(* CODESYS project unilib.library
   Company: Beckhoff Automation GmbH & Co. KG
   DefaultNamespace: TC3_UniLib
   Version: 1.2.10.2
   Placeholder: UniLib Gruppe 11
   Author: Christian Frickenstein, Bernhard Edenfeld, Benedikt Daut
   Description: Zentrale Bausteine für die Programmierung in der Gruppe 11. Hinweise zu den Versionsnummern: 1. Zahl: Grundsätzliche Version für TwinCAT3, 2. Zahl: für die verschiedenen Varianten. Nicht abwärtskompatibel, 3. Zahl: Neue Bausteine oder Funktionen hinzugefügt, aber abwärtskompatibel ggf. neue Eingänge oder Umbenennungen. 4. Zahl: Bugfixes, bedingungslos abwärtskompatibel
   Title: UniLib Gruppe 11

Project tree, tasks and I/O mapping:
  libraries: Tc2_EtherCAT, * (Beckhoff Automation GmbH); Tc2_IoFunctions, * (Beckhoff Automation GmbH); Tc2_MC2, * (Beckhoff Automation GmbH); Tc2_MC2_Drive, * (Beckhoff Automation GmbH); Tc2_SerialCom, * (Beckhoff Automation GmbH); Tc2_Standard, * (Beckhoff Automation GmbH); Tc2_System, * (Beckhoff Automation GmbH); Tc2_Utilities, * (Beckhoff Automation GmbH); Tc3_JsonXml, * (Beckhoff Automation GmbH); Tc3_Module, * (Beckhoff Automation GmbH)
  DUTs/
    ComPort/
      data type E_ComPortHardware
      data type E_ComPortKlemmenBytes
      data type E_ComPortProtokoll
      data type ST_ComPortFlags
      data type ST_ComPortInData
      data type ST_ComPortIntBuffer
      data type ST_ComPortOptions
      data type ST_ComPortOptionsIntern
      data type ST_ComPortOutData
      data type ST_ComPortStringBuffer
      data type ST_InInfoDataSerielleKlemme
      data type ST_MethodResult
    DiagEL2904/
      data type ST_EL2904Diag
      data type ST_EL2904Temp
    EAP/
      data type ST_EAP_Kommunikation
      data type ST_EAP_Receive
      data type ST_EAP_Send
      data type ST_StepCtrl
      data type ST_StepPara
      data type ST_TEMP_EAP_TEST
      data type ST_TempEAPDaten
      data type ST_TwinSAFE_Connection
      data type U_EAP_Kommunikation
    HMI_DataExchange/
      data type ST_HMIDataExchange
    HMI_Grundstrukturen/
      data type ST_HandFktHMI
      data type ST_OP_HMI
      data type ST_OP_Visual
    HMI_Meldungen/
      Meldelisten/
        Allgemein/
          data type ST_MeldTextAllgm
        InternAchsen/
          data type ST_MeldAchsfehler
          data type ST_MeldAchsGruppe
        InternEinspeis/
          data type ST_MeldAuffrischKlemme
          data type ST_MeldEinspeisKlemme
        InternSafety/
          data type ST_MeldKlemme
          data type ST_MeldSafetyFBErrors
          data type ST_MeldSafetygruppe
          data type ST_MeldSafetyOuts
        InternSchaltschrank/
          data type ST_MeldElektrSichg
          data type ST_MeldKlimaGeraet
          data type ST_MeldMotSchutzS
          data type ST_MeldSchaltNetzT
          data type ST_MeldSichgAutom
          data type ST_MeldThermoUeberw
          data type ST_MeldUSV
        InternSchutzbereich/
          data type ST_MeldNotHalt
          data type ST_MeldSchutzbereichOffen
          data type ST_MeldSichLichtg
          data type ST_MeldStHLuft
          data type ST_MeldTuerFrgBremsentest
          data type ST_MeldWartgTuer
        InternSonstiges/
          data type ST_MeldADS_ExchangeError
          data type ST_MeldADSKommError
          data type ST_MeldBetriebsdruck
          data type ST_MeldDatenanf
          data type ST_MeldEAPKommError
          data type ST_MeldEtherCAT
          data type ST_MeldGrundstellung
          data type ST_MeldIOLinkKlemme
        UniAnstg/
          data type ST_MeldAchsKontrl
          data type ST_MeldTextUniAchs
          data type ST_MeldTextUniAktr
          data type ST_MeldTextUniAntr
          data type ST_MeldTextUniWkzg
          data type ST_MeldTextUniZyli
        data type ST_MeldAchsList
        data type ST_MeldEAPList
        data type ST_MeldIOLinkList
        data type ST_MeldKommunikationsList
        data type ST_MeldPotentialList
        data type ST_MeldSafetyList
        data type ST_MeldSchaltSchrList
        data type ST_MeldSchutzberList
        data type ST_MeldSeriellComPort
      data type ST_0100_Meldungen
      data type ST_ParamHMIMaschine_Beispiel
    HMI_Parameter/
      data type ST_UniAchsAnstgParam
      data type ST_UniAntrAnstgParamAggr
      data type ST_UniAntrAnstgParamAggrHF
      data type ST_UniAntrAnstgParamTrsp
    HMI_UniAnstgHandFktMeldungen/
      data type E_AnstgArtUniAktr
      data type E_AnstgArtUniAntr
      data type E_AnstgArtUniWkzg
      data type E_AnstgArtUniZyli
      data type E_AntriebTyp
      data type E_ZylinderTyp
      data type ST_UniAchsAnstg
      data type ST_UniAktrAnstg
      data type ST_UniAntrAnstg
      data type ST_UniBaustein
      data type ST_UniGrdstlgAbl
      data type ST_UniWkzgAnstg
      data type ST_UniZyliAnstg
    Meldebox/
      data type ST_MessageBox
    NcAchsen/
      data type ST_AchsAuftrg
      data type ST_AchsFreigb
      data type ST_AchsGrdfkt
      data type ST_AchsInOut
      data type ST_AchsKoppln
      data type ST_AchsMeldg
      data type ST_AchsParam
      data type ST_AchsStatus
      data type ST_NcAchsen
    SEW/
      data type ST_SEWInput
      data type ST_SEWOutput
    TwinSAFE/
      data type E_SafetyType
      data type ST_TwinSAFE_Conn_Info
      data type ST_TwinSAFE_ConnInfoBasis
      data type ST_TwinSAFE_FB_Info
      data type ST_TwinSAFE_Group_Info
      data type ST_TwinSAFEConnInfo4Byte
      data type ST_TwinSAFEConnInfo5Byte
      data type ST_TwinSAFEKlemmenInfo
    data type ST_TimeStamp
    data type ST_TimeStruct
  GVLs/
    global variables AllgemeineParameter
    global variables ComPortParameterliste
    global variables GlobalVar_Allgemein
    global variables GlobalVar_Farben
    global variables GlobalVar_TestMeld
  POUs/
    ComPort_2_0_1_0/
      function F_ComReceiveBarcode [ST]
      function F_ComSendBarcode [ST]
      function block FB_ComBackground [ST]
      function block FB_ComConfig [ST]
      function block FB_ComMain [ST]
      function block FB_ComPortOld [ST]
    ComPort_3_0_1_0/
      function block FB_ComPort [ST]: ccl_Backround, ccl_Main, ccl_Messages, ccl_Receive, FB_init, nccl_Config, nccl_PrepareSendBarcode, nccl_ReceiveBarcode, nccl_Reset, nccl_Send, P_bDatenVorhanden, P_stEmpfangeneDaten, P_stEmpfangenerString
      data type ST_MeldComPort
    DiagSafety/
      function block FB_DiagEL2904 [ST]: act_Diag, act_DiagObjekte
      function block FB_DiagEL2912 [ST]: act_Diag
      function block FB_TwinSAFE_Conn_Info [ST]: act_Diag, act_State, actInfo
      function block FB_TwinSAFE_FBs_Info [ST]: act_Diag, act_State, actInfoAND, actInfoConnectionShutDown, actInfoDecoupler, actInfoEDM, actInfoEStop, actInfoMON, actInfoMuting, actInfoOPMode, actInfoOR, actInfoRS, actInfoSR, actInfoTOF, actInfoTON, actInfoTwoHand
      function block FB_TwinSAFE_Group_Info [ST]: act_State, actInfo
      function block FB_TwinSAFEConnInfo [ST]: act_Diag, act_State, actInfo
      function block FB_TwinSAFEConnInfo4Byte [ST]: a_Info, b_State, c_Diag
      function block FB_TwinSAFEConnInfo4Byte_1 [ST]: a_Info, b_State, c_Diag
      function block FB_TwinSAFEConnInfo5Byte [ST]: a_Info, b_State, c_Diag
      function block FB_TwinSAFEConnInfo5Byte_1 [ST]: a_Info, b_State, c_Diag
      function block FB_TwinSAFEConnInfoBasis [ST]: a_Info, b_State, c_Diag
      function block FB_TwinSAFEFBsInfo [ST]: act_Diag, act_State, actInfoAND, actInfoConnectionShutDown, actInfoDecoupler, actInfoEDM, actInfoEStop, actInfoMON, actInfoMuting, actInfoOPMode, actInfoOR, actInfoRS, actInfoSR, actInfoTOF, actInfoTON, actInfoTwoHand
      function block FB_TwinSAFEGroupInfo [ST]: act_State, actInfo
      function block FB_TwinSAFEKlemmeInfo [ST]: a_Initialisierung, b_Ablauf, c_EL6900, c_EL6910, d_EK1914, d_EL1904, d_EL1918, d_EP1908, d_EP1918, d_EP1957, e_EL2904, e_EL2911, e_EL2912, e_EP2918, f_AX5805, f_AX5806
    Diverse/
      function F_Skalierung [ST]
      function F_Switchbyte [ST]
      function block FB_Blinker [ST]
      function block FB_ElectronicFuseIOLink [ST]: a_GetCurrent, b_GetStatus, z_Message, z_Output
      function block FB_SafetyElementAnz [ST]
      function block FB_UsvStatus [ST]
      function block FB_WartgTuer [ST]: a_TuerEntrieg, b_AutomHalt
      function block FB_WartgTuerMeld [ST]: a_TuerEntrieg, b_AutomHalt, z_Meld
      function block FB_WartgTuerMeldAnz [ST]: a_TuerEntrieg, b_AutomHalt, c_Anzeige, z_Meld
    EAP/
      function block FB_EAP_Kommunikation [ST]: _00_Init, _02_TwinSAFE, m_DatenBereitstellen, m_Receive, m_Send, m_Senden
      function block FB_EAP_Kommunikation_V2 [ST]: _02_TwinSAFE, _07_Senden_Empfangen, _10_Meldungen, m_Senden
      function block FB_StepUebw [ST]
    EtherCATDiagnose/
      data type E_EcCommState
      function block FB_EtherCATDiag [ST]: a_GetSlaveAdresses, b_GetSlaveStates, c_GetTopoDataLen, d_GetTopoData, e_ScanSlaves, f_GetSlaveIdentity, g_GetSlaveName, h_GetScannedSlaveName, i_ErrorMessage, j_CheckMasterDevState, k_SlaveErrorMessage
      function block FB_EtherCATFrameDiag [ST]
      function block FB_IoLinkFehler [ST]
      data type ST_EcMasterDevState
      data type ST_EcPortAddr
      data type ST_SlaveState
      data type ST_SlaveStateInfo
      data type ST_SlaveStateInfoScanned
      data type ST_TopologyData
    Grundstellung/
      function block FB_UniGrdstlgAbl [ST]: a_AnAbwahl, b_StepAblauf, y_ZustAnzg, z_HinwMeld
      function block FB_UniGrdstlgAblBereich [ST]: a_AnAbwahl, b_StepAblauf, y_ZustAnzg, z_HinwMeld
      function block FB_UniGrdstlgAblGesamt [ST]: a_AnAbwahl, b_StepAblauf, y_ZustAnzg, z_HinwMeld
    Logging/
      function F_AdsErrorIdToString [ST]
      function F_TimeStruct [ST]
      function block FB_LogToFile [ST]
      function block FB_StepHistory [ST]
      function block FB_TaktzeitAuswert [ST]: a_DateiSchreiben
    MeldTest/
      function block FB_MeldTestAllgemein [ST]
    Time/
      function block FB_Zeitstempel [ST]
    UniBausteine/
      function block FB_LaufzMeldg [ST]
      function block FB_LaufzMeldgAktr [ST]
      function block FB_UniAchsAnstg [ST]: a_Standard, w_InOutNc, y_ZustAnzg, z_FehlMeld
      function block FB_UniAktrAnstg [ST]: a_Standard, x_AusgZuw, y_ZustAnzg, z_FehlMeld
      function block FB_UniAntrAnstg [ST]: a_Aggregat, b_Transport, c_Verstellg, x_AusgZuw, y_ZustAnzg, z_FehlMeld
      function block FB_UniAntrAnstgSEW [ST]: a_Aggregat, b_Transport, c_Verstellg, d_EilSchleich, u_AggEinlZykl, v_AggBetrZykl, w_InOutSEW, x_AusgZuw, y_ZustAnzg, z_FehlerAusw, z_FehlMeld
      function block FB_UniAntrAnstgSEW_IO [ST]: a_Aggregat, b_Transport, c_Verstellg, d_EilSchleich, u_AggEinlZykl, v_AggBetrZykl, w_InOutSEW, x_AusgZuw, y_ZustAnzg, z_FehlMeld
      function block FB_UniHydrAnstgHubb [ST]: a_Standard, x_AusgZuw, y_ZustAnzg, z_FehlMeld
      function block FB_UniWkzgAnstg [ST]: a_Standard, b_PulsUebw, x_AusgZuw, y_ZustAnzg, z_FehlMeld
      function block FB_UniZyliAnstg [ST]: a_Standard, b_MittelStellung, c_TestMode, x_AusgaengeZuweisen, y_ZustaendeAnzeigen, z_FehlerMeldung
*)

// DUTs/ComPort/E_ComPortHardware
{attribute 'qualified_only'}
// Comportdefinition der Hardware
TYPE E_ComPortHardware:(
	cComportPc,	// Der Comport kommt aus einem PC
	cComportKL,	// Der Comport kommt von einer KL-Klemme
	cComportEL	// Der Comport kommt von einer EL-Klemme
);
END_TYPE

// DUTs/ComPort/E_ComPortKlemmenBytes
{attribute 'qualified_only'}
// Größe des Byte-Streams aus der Hardware-Verbindung
TYPE E_ComPortKlemmenBytes:(
	cComport3Bytes,	// Der Komport liefert einen Byte-Stream von 3 Byte, alte Klemmen
	cComport5Bytes,	// Der Komport liefert einen Byte-Stream von 5 Byte, alte Klemmen
	cComport22Bytes	// Der Komport liefert einen Byte-Stream von 22 Byte, aktueller Standard
);
END_TYPE

// DUTs/ComPort/E_ComPortProtokoll
{attribute 'qualified_only'}
// Protokoll, wie der empfangene Byte-Stream ausgewertet werden soll
TYPE E_ComPortProtokoll :(
	cProtokollNone,	// Protokoll, wie der Byte-Stream ausgewertet werden soll. Hier wird der Byte-Stream dirket ausgegeben
	cProtokollData,	// Protokoll, wie der Byte-Stream ausgewertet werden soll. Hier wird der Byte-Stream dirket ausgegeben
	cProtokollDirect,	// Protokoll, wie der Byte-Stream ausgewertet werden soll. Hier wird der Byte-Stream dirket ausgegeben
	cProtokollBarcode,	// Protokoll, wie der Byte-Stream ausgewertet werden soll. Hier wird der Byte-Stream als STRING ausgegeben
	cProtokollP3964	// Protokoll, wie der Byte-Stream ausgewertet werden soll. Hier wird der Byte-Stream im P3964-Format ausgegeben
);
END_TYPE

// DUTs/ComPort/ST_ComPortFlags
TYPE ST_ComPortFlags :
STRUCT
	(* Konfiguration *)
	bConfigFlag		: BOOL;			(* Anstossen der Schnittstellenkonfiguration *)

	(* Schnittstellenpuffer loeschen *)
	bResetFlag		: BOOL;			(* Loeschen des internen Schnittstellenpuffers *)

	(* Empfangen *)
	bRxFlag			: BOOL;			(* Anstossen der Datenauswertung bei Empfang *)
	bWaitQuitFlag	: BOOL;			(* Quittieren der neg. Flanke von VB*)

	(* Senden *)
	bTxFlag			: BOOL;			(* Anstossen des Sendens *)
END_STRUCT
END_TYPE

// DUTs/ComPort/ST_ComPortInData
// Datentyp für die Verbindung zur Hardwareschnittstelle. Für alle Byte-Streamtypen. Nur eine Verbindung nutzen!!!
TYPE ST_ComPortInData :
STRUCT
	stKlemmeIn3B	: Tc2_SerialCom.KL6inData;	// Inputdaten für 3Byte-Klemmen
	stKlemmeIn5B	: Tc2_SerialCom.KL6inData5B;	// Inputdaten für 5Byte-Klemmen
	stKlemmeIn22B	: Tc2_SerialCom.KL6inData22B;	// Inputdaten für 22Byte-Klemmen
	stPCIn			: Tc2_SerialCom.PcComInData;	// Inputdaten für PC-Verbindung
	stInfoData		: ST_InInfoDataSerielleKlemme;	// Infodaten, sollten mit einer Klemme verküpft werden um sie automatisch zu parametrieren
END_STRUCT
END_TYPE

// DUTs/ComPort/ST_ComPortIntBuffer
// Datentyp für den Internen Byte-Stream
TYPE ST_ComPortIntBuffer :
STRUCT
	arrData	: ARRAY [0..cBufferSize_IntBuffer] OF UINT;	// Interner Puffer für die Empfangenen Bytes
END_STRUCT
END_TYPE

// DUTs/ComPort/ST_ComPortOptions
// Optionen für den Comport
TYPE ST_ComPortOptions:
STRUCT
	nId				: UINT;	// Allgemeine Nummerierung
	
	nBaudrate  		: UINT;	// 1200, 2400, 4800, 9600, 19200
	nDatenbits		: UINT;	// 7, 8
	nStopbits 		: UINT;	// 1, 2
	nParitaet 		: INT;	// 0: keine Parität, 1: gerade(even) Parität, 2: ungerade(odd) Parität
	nHandshake		: INT;	// 0: Kein Handshake, 1: RTS/CTS, 2: XON/XOFF
	
	eProtokoll 		: E_ComPortProtokoll;	// 0: kein, 1: Daten, 2: Direkt, 3: Barcode, 4: 3964
	nPrefix 			: UINT;	// 0: kein, 2: STX
	nSuffix1 		: UINT;	// 0: kein, 13: CR, 3: ETX, 4: EOT 
	nSuffix2 		: UINT;	// 0: kein, 10: LF
	nTimeout 		: UINT;	// Maximale Zeit zwischen zwei Zeichen, bei String oder Barcodeempfang
	nLength			: INT;	// Anzahl der zu empfangenen Zeichen, incl. Präfix und Suffix
	
	ePort				: E_ComPortHardware;	// 0: PC, 1: Klemme, 2: E-Klemme
	eComPortBytes	: E_ComPortKlemmenBytes;	// 0: 3 Bytes, 1: 5 Bytes, 2: 22 Bytes
	nAktiv			: UINT;	// 0: Schnittstelle nicht aktiv, 1: Schnittstelle aktiv
	nCommVB			: UINT;	// 0: DotNet als Applikation, 1: VisualBasic als Applikation
END_STRUCT
END_TYPE

// DUTs/ComPort/ST_ComPortOptionsIntern
// Datentyp für die Internen Optionen
TYPE ST_ComPortOptionsIntern :
STRUCT
	nPrefix			: BYTE;	// Präfix als ASCII-Zeichen
	sPrefix			: STRING(10);	// Präfix als String
	nLenPrefix		: BYTE;	// Länge des Prefixes

	arrSuffix		: ARRAY[1..2] OF BYTE;	// Suffix als ASCII-Array
	sSuffix			: STRING(10);	// Suffix als String
	nLenSuffix		: BYTE;	// Länge des Suffixes

	tTimeTimeout	: TIME;	// Maximale Zeit zwischen zwei Zeichen, bei String oder Barcodeempfang
   nLength			: INT;	// Anzahl der zu empfangenen Zeichen, incl. Präfix und Suffix
END_STRUCT
END_TYPE

// DUTs/ComPort/ST_ComPortOutData
// Datentyp für die Verbindung zur Hardwareschnittstelle. Für alle Byte-Streamtypen. Nur eine Verbindung nutzen!!!
TYPE ST_ComPortOutData :
STRUCT
	stKlemmeOut3B	: KL6outData;	// Outputdaten für 3Byte-Klemmen (obsolet)
	stKlemmeOut5B	: KL6outData5B;	// Outputdaten für 5Byte-Klemmen	(obsolet)
	stKlemmeOut22B	: KL6outData22B;	// Outputdaten für 22Byte-Klemmen (standard)
	stPCOut			: PcComOutData;	// Outputdaten für PC-Verbindungen
END_STRUCT
END_TYPE

// DUTs/ComPort/ST_ComPortStringBuffer
// Datentyp: Empfangener Stream als STRING in variabler Größe
TYPE ST_ComPortStringBuffer :
STRUCT
	sData	: STRING(cBufferSize_StringBuffer);	// variable STRING-Variable
END_STRUCT
END_TYPE

// DUTs/ComPort/ST_InInfoDataSerielleKlemme
// Datentyo zur ADS-Verbindung mit der Klemme
TYPE ST_InInfoDataSerielleKlemme :
STRUCT
	stADSNetId	: Tc2_System.T_AmsNetIdArr;	// ADS-NETID 172.50.12.1.1.1 oder ähnlich
	nADSPort		: UINT;	// ADS-Port: 1002 oder höher
END_STRUCT
END_TYPE

// DUTs/ComPort/ST_MethodResult
// Ergebnisvariable einer Methode
TYPE ST_MethodResult :
STRUCT
	bBusy		: BOOL;	// Methode ist aktiv und noch nicht abgearbeitet
	bDone		: BOOL;	// Methode ist abgearbeitet
	bError	: BOOL;	// Error bei Bearbeitung aufgetreten 
	nErrorId	: INT;	//	Error als ID
	sError	: STRING;	// Error als Klartext
END_STRUCT
END_TYPE

// DUTs/DiagEL2904/ST_EL2904Diag
// OBSOLET, wenn man FB_TwinSAFEKlemmenInfo benutzt
TYPE ST_EL2904Diag :
STRUCT
	nDummyData1								:ARRAY[0..10] OF UINT;

(* Error at the outputs *)
	nErrorOutputs							:UINT;

(* Supply error *)
	nSupplyError							:UINT;

(* Temperature error *)
	nTemperatureError						:UINT;

	nDummyData2								:ARRAY[0..1] OF UINT;

END_STRUCT
END_TYPE

// DUTs/DiagEL2904/ST_EL2904Temp
// OBSOLET, wenn man FB_TwinSAFEKlemmenInfo benutzt
TYPE ST_EL2904Temp :
STRUCT	
	nInternalTemperature1					:INT;	(* Temperature 1 [°C] *)
	nInternalTemperature2					:INT;	(* Temperature 2 [°C] *)
	nInternalTemperatureOutputs			:INT;	(* Temperature 2 [°C] *)
END_STRUCT
END_TYPE

// DUTs/EAP/ST_EAP_Kommunikation
{attribute 'pack_mode' := '0'}
TYPE ST_EAP_Kommunikation :
STRUCT
	KommBits				: DWORD;
	TeilID				: STRING(19);
	TeilStatus			: DWORD;		
	ZusatzInfo1			: DWORD;		
	ZusatzInfo2			: DWORD;		
	ZusatzInfo3			: DWORD;		
	ZusatzInfo4			: DWORD;		
	ZusatzInfo5			: DWORD;		
	ZusatzInfo6			: DWORD;		
	ZusatzInfo7			: DWORD;		
	ZusatzInfo8			: DWORD;		
	ZusatzInfo9			: DWORD;		
	ZusatzInfo10		: DWORD;		
	
	//71BYTE

END_STRUCT
END_TYPE

// DUTs/EAP/ST_EAP_Receive
TYPE ST_EAP_Receive :
STRUCT
	VarState		AT %I* : UINT;
	Quality		AT %I* : UINT;
	CycleIndex	AT %I* : UINT;
	VarData		AT %I* : U_EAP_Kommunikation; 
END_STRUCT
END_TYPE

// DUTs/EAP/ST_EAP_Send
TYPE ST_EAP_Send :
STRUCT
	FrameState	AT %I* : UINT;
	FrameCtrl	AT %Q* : UINT;
	VarState		AT %I* : UINT;
	VarCtrl		AT %Q* : UINT;
	VarData		AT %Q* : U_EAP_Kommunikation; 
END_STRUCT
END_TYPE

// DUTs/EAP/ST_StepCtrl
// SK20190724:
// StepControl entählt folgende Funktionalitäten:
//	-> Delayabfrage und -Ausgabe
//	-> fbStepHistory mit optionaler Status Eintragung
//	-> Variablen für die Schrittkette
// !!! <VarName>.fbHistory(IQ_StepPara := <VarName>.IQ); notwendig
TYPE ST_StepCtrl :
STRUCT
	IQ				: ST_StepPara;
	fbHistory	: FB_StepUebw;
END_STRUCT
END_TYPE

// DUTs/EAP/ST_StepPara
TYPE ST_StepPara :
STRUCT
	
	nStep			: INT;
	sStatus		: T_MaxString;
	I_tDelay		: TIME;		// Delayvorgabe			Timer läuft ab, wenn Step = oldStep
	Q_bDelay		: BOOL;		// Delay abgelaufen
	I_bAblaufIN	: BOOL;		//								Timer läuft ab, wenn I_bAblaufIN = TRUE
	I_tAblauf	: TIME;		// Delayvorgabe
	Q_bAblauf	: BOOL;		// Delay abgelaufen
	I_bReset		: BOOL;
	I_bSaveLog	: BOOL;

END_STRUCT
END_TYPE

// DUTs/EAP/ST_TEMP_EAP_TEST
TYPE ST_TEMP_EAP_TEST :
STRUCT
	tonStartDif			: TON;
	tonDifEAP			: TON;
	tonDifKabel			: TON;
	
	bStartDifEAP		: BOOL;
	bStartDifKabel		: BOOL;
	
	ftStartDif			: F_TRIG;
	ftStartEAP			: F_TRIG;
	ftStartKabel		: F_TRIG;
	rtStopMessung		: R_TRIG;

	
	bEAPSchneller		: BOOL;
	bKabelSchneller	: BOOL;
	bGleich				: BOOL;
	bAlleUnngleich		: BOOL;
	tZeitDif				: TIME;
	
	nEAPkeinSignal		: INT;	
	
	
	

END_STRUCT
END_TYPE

// DUTs/EAP/ST_TempEAPDaten
TYPE ST_TempEAPDaten :
STRUCT
	sTeilenummer		: STRING(19);	// Teilenummer 
	wStatus				: DWORD;			// Der Status des Teils
	wZusatzinfo1		: DWORD;			//	Zusätzliche Infos 1
	wZusatzinfo2		: DWORD;			// Zusätzliche Infos 2
	wZusatzinfo3		: DWORD;			// Zusätzliche Infos 3
	wZusatzinfo4		: DWORD;			// Zusätzliche Infos 4
	wZusatzinfo5		: DWORD;			// Zusätzliche Infos 5
	wZusatzinfo6		: DWORD;			// Zusätzliche Infos 6
	wZusatzinfo7		: DWORD;			// Zusätzliche Infos 7
	wZusatzinfo8		: DWORD;			// Zusätzliche Infos 8
	wZusatzinfo9		: DWORD;			// Zusätzliche Infos 9
	wZusatzinfo10		: DWORD;			// Zusätzliche Infos 10
END_STRUCT
END_TYPE

// DUTs/EAP/ST_TwinSAFE_Connection
TYPE ST_TwinSAFE_Connection :
STRUCT
	 
	I_nID				: INT;
	I_sConnName		: STRING;
	I_nGroupID		: INT;
	Q_bIn0			: BOOL;
	Q_bIn1			: BOOL;
	Q_bIn2			: BOOL;
	Q_bIn3			: BOOL;
	Q_bIn4			: BOOL;
	Q_bIn5			: BOOL;
	Q_bIn6			: BOOL;
	Q_bIn7			: BOOL;
	Q_bOut0			: BOOL;
	Q_bOut1			: BOOL;
	Q_bOut2			: BOOL;
	Q_bOut3			: BOOL;
	Q_bOut4			: BOOL;
	Q_bOut5			: BOOL;
	Q_bOut6			: BOOL;
	Q_bOut7			: BOOL;
	Q_bErrDiag		: BOOL;
	Q_bErrState		: BOOL;
	Q_sDiag			: STRING(255);
	Q_sState			: STRING(255);

END_STRUCT
END_TYPE

// DUTs/EAP/U_EAP_Kommunikation
TYPE U_EAP_Kommunikation :
UNION
	Komm	: ARRAY[1..71] OF BYTE;
	Data	: ST_EAP_Kommunikation;
END_UNION
END_TYPE

// DUTs/HMI_DataExchange/ST_HMIDataExchange
{attribute 'pack_mode' := '1'}
// TODO: muss in die BAAvalonLib wandern

TYPE ST_HMIDataExchange :
STRUCT
	bNewData			: BOOL;		// Trigger Variable Plc setzt = TRUE => Oberfläche setzt zurück (FALSE)
	nStatus			: DINT;		// 1 Ok / > 1 Fehler
	sData				: STRING;	// Daten die von Plc kommen Barcode, Bohrbilder, PersonalNummern
	nTyp				: INT;		// Zur weitern Differenzierung der Daten (z.B. 1:Teilebarcode/2:Stapelbarcode)
	sSource			: STRING;	// Quelle von der die Daten kommen ggf. zu weiteren Auswertung in der Obefläche
  	sDestination	: STRING;	// Ziel mit dem die Daten in der Oberfläche ausgewertet werden
END_STRUCT
END_TYPE

// DUTs/HMI_Grundstrukturen/ST_HandFktHMI
// Handfunktion in der Oberfläche. Wird in den UniBausteinen verwendet.
// Diese Struktur hat immer nur eine Taste/Schalter
// Es gibt zwei verschiedene Auslesevarianten
// 1. Variante: mit Kommentaren. Vorteil: Einzeiler, altbekannt, wirkt simpler; Nachteil: Keine Änderung bei Online-Change
// 2. Variante: mit Attributen. Vorteil: Namensänderungen werden bei Online-Change übernommen
// Beispiel 1. Variante:
// arrManFunction	: ARRAY[1..3] OF ST_HandFktHMI; (*@1: Zylinder @2:1 Belegung @3:2 Test @4:5 Hand*)	@2-@9 sind die Tasten/Schalter. Die Zahl hinter dem Doppelpunkt ist der Eingabetyp
// @2:1 ist ein Taster; @2:2 ist ein Schalter; @2:3 noch nicht implementiert; @2:4 noch nicht implementiert; @2:5 Eingabemöglichkeit als Text (sImage)
// Beispiel 2. Variante:
// {attribute 'MaschPara.Name' := 'HandTest'}
// {attribute 'MaschPara.Handfunktion.Btn1' := '2 Belegung'}
// {attribute 'MaschPara.Handfunktion.Btn2' := '1 Test}
// {attribute 'MaschPara.Handfunktion.Btn3' := '2 Hand'}
// arrManFunction	: ARRAY[1..3] OF ST_HandFktHMI;
// TODO: muss in die BAAvalonLib wandern

{attribute 'pack_mode' := '1'}
TYPE ST_HandFktHMI :
STRUCT
	bySwitch			:BYTE;	// Bei Betätigung wird Bit0 TRUE. Man kann auch >0 abfragen
	byStatus			:BYTE;	// mit Bit 0 wird die Taste gesperrt
	iDisplayMode	:INT;		// Blinkmode der einzelnen Tasten: 0= normale Farbe kein blinken, 1= langsam blinken, 2= schnell blinken, 3= noch nicht implementiert
	sText				:STRING;	// Text der einzelnen Tasten
	sColour			:STRING;	// Farbe der einzelnen Tasten in 16#XXXXXXXX aber ohne 16#
	sImage			:STRING;	// Wert vom Typ5 der Eingabemöglichkeit. Für die SVG-Dateien einfach 'Dateiname.svg' eingeben
END_STRUCT
END_TYPE

// DUTs/HMI_Grundstrukturen/ST_OP_HMI
// Strukturierung einer Station zur Anzeige in der 2D Übersicht.
// Hat maximal 10 Taster/Schalter/Icons
// Beispiel zur Implementierung
// In der 3D-Übersicht ist die STRING-Var 'Name' der Name des Buttons mit dem man zu dieser Struktur kommt.
// In der Tree-View-Übersicht ist 'MaschPara.Name' der Name in den Layers/Knoten 
//	{attribute 'MaschPara.Name' := 'Maschinenteil PXYZ'}
//	stStatus	: ST_OP_HMI;
// TODO: muss in die BAAvalonLib wandern

{attribute 'pack_mode' := '1'}
TYPE ST_OP_HMI :
STRUCT
	Name				:STRING;	// Name der Station, die in der 3D-Ansicht als Buttonbeschreibung angezeigt wird.
	
	BtnSignal		:ARRAY[1..10] OF BOOL;			// hiermit kann der Zustand des Tasten/Schalter 1-10 ausgelesen werden.
	BtnEnable		:ARRAY[1..10] OF BOOL;			// hiermit können die Tasten/Schalter 1-10 angezeigt.
	BtnColor			:ARRAY[1..10] OF STRING(8);	// Farbe der einzelnen Tasten in 16#XXXXXXXX aber ohne 16#
	BtnText			:ARRAY[1..10] OF STRING;		// Text der einzelnen Tasten
	BtnPicture		:ARRAY[1..10] OF STRING;		// Pfad zum Icon der einzelnen Tasten. Für die SVG-Dateien einfach 'Dateiname.svg' eingeben
	BtnDisplayMode	:ARRAY[1..10] OF INT;			// Blinkmode der einzelnen Tasten: 0= normale Farbe kein blinken, 1= langsam blinken, 2= schnell blinken, 3= noch nicht implementiert
   StatusText  	:ARRAY[1..10] OF STRING(255);	// Statustext

	StepNr      	:INT;		// aktueller Schritt in dem sich die Bearbeitung der Station befindet
	StatusPicture1 :STRING;	// Pfad zu einem Icon/Bild Für die SVG-Dateien einfach 'Dateiname.svg' eingeben
	StatusPicture2 :STRING; // Pfad zu einem Icon/Bild Für die SVG-Dateien einfach 'Dateiname.svg' eingeben
	InfeedReady    :BOOL;	// Transportzustand als LED-Icon: Eintransport bereit
	InfeedActive   :BOOL;	// Transportzustand als LED-Icon: Eintransport aktiv
	InfeedFinished :BOOL;	// Transportzustand als LED-Icon: Eintransport fertig
	OutfeedReady  	:BOOL;	// Transportzustand als LED-Icon: Austransport bereit
	OutfeedActive	:BOOL;	// Transportzustand als LED-Icon: Austransport aktiv
	OutfeedFinished:BOOL;	// Transportzustand als LED-Icon: Austransport fertig
	StatusColor		:STRING(8);	// Statusfarbe als String in HEX 16#XXXXXXXX aber ohne 16#
END_STRUCT
END_TYPE

// DUTs/HMI_Grundstrukturen/ST_OP_Visual
// Strukturierung eines Anzeigeelements in der 2D Übersicht.
// Das Attribut mit 'Typ' muss immer mitdeklariert sein. Auch wenn es leer ist und keine Funktion hat.
// Beispiel zur Implementierung:
//	{attribute 'MaschPara.Name' := 'DigitalerSensor'}
//	{attribute 'MaschPara.Typ' := ''}
//	stSensorDigital	: ST_OP_Visual;
// TODO: muss in die BAAvalonLib wandern

{attribute 'pack_mode' := '1'}
TYPE ST_OP_Visual :
STRUCT
	bIsChecked		: BOOL;		// Zustand des Visu-Elements
	bIsEnabled		: BOOL	:= TRUE;		// FALSE = ausgegraut
	iDisplayMode	: INT;		// Blinkmode: 0= normale Farbe kein blinken, 1= langsam blinken, 2= schnell blinken, 3= noch nicht implementiert
	sText				: STRING;	// Text des Visu-Elements
	sColour			: STRING;	// Farbe im Format: 16#XXXXXXXX aber ohne 16#
	sImage			: STRING	:= 'OP_States\Door.png';	// Pfad zu einem Icon/Bild. Für die SVG-Dateien einfach 'Dateiname.svg' eingeben
END_STRUCT
END_TYPE

// DUTs/HMI_Meldungen/Meldelisten/Allgemein/ST_MeldTextAllgm
// Diese Struktur stellt eine allgemeine Meldung dar. Es kann zwischen Hinweis, Warnung und Fehler gewählt werden.
// Es muss immer ein kompletter Meldetext mit angegeben werden.
{attribute 'pack_mode' := '1'}
TYPE ST_MeldTextAllgm :
STRUCT
	 
{attribute 'Message.SourceID'}
	SourceID			:DINT;
	
{attribute 'Message.SourceName'}
   SourceName		:STRING;
 
{attribute 'Message.Text' := '%Var1'}		
{attribute 'Message.Info' := '%Var2'}
{attribute 'Message.Type' := '1'}	
{attribute 'Message.Log'  := '1'}
{attribute 'Message.Var1' := 'sText'} 
{attribute 'Message.Var2' := 'sInfo'}  
	bMeldAusg			:BOOL;	
 
{attribute 'Message.Text' := '%Var1'}		
{attribute 'Message.Info' := '%Var2'}
{attribute 'Message.Type' := '4'}	
{attribute 'Message.Log'  := '1'}
{attribute 'Message.Var1' := 'sText'}   
{attribute 'Message.Var2' := 'sInfo'}  
	bWarnAusg			:BOOL;	
 
{attribute 'Message.Text' := '%Var1'}		
{attribute 'Message.Info' := '%Var2'}
{attribute 'Message.Type' := '7'}	
{attribute 'Message.Log'  := '1'}
{attribute 'Message.Var1' := 'sText'}   
{attribute 'Message.Var2' := 'sInfo'}  
	bFehlAusg			:BOOL;	
 
{attribute 'Message.Text' := '%Var1'}		
{attribute 'Message.Info' := '%Var2'}
{attribute 'Message.Type' := '8'}	
{attribute 'Message.Log'  := '1'}
{attribute 'Message.Var1' := 'sText'}   
{attribute 'Message.Var2' := 'sInfo'}  
	bKritFehlerAusg	:BOOL;	

	sText		:T_MaxString;	// z.B. Fehlermeldungen
	sInfo		:T_MaxString;	// ggf. BMK
	
END_STRUCT
END_TYPE

// DUTs/HMI_Meldungen/Meldelisten/InternAchsen/ST_MeldAchsfehler
{attribute 'pack_mode' := '1'}
TYPE ST_MeldAchsfehler :
STRUCT
{attribute 'Message.SourceID'}
	SourceID				:DINT;
	
{attribute 'Message.SourceName'}
   SourceName			:STRING	:= 'Achsfehler';

	
{attribute 'Message.Text' := 'Achsfehler: Freifahren erforderlich! Bitte Service-Taste betätigen !'}		
{attribute 'Message.Info' := '%Var1'}
{attribute 'Message.Type' := '8'}	
{attribute 'Message.Log'  := '1'}
{attribute 'Message.Var1' := 'sBMK'}  	
	bMeldFreifahren	:BOOL;	
	
{attribute 'Message.Text' := 'Achsfehler: Reset erforderlich! Bitte Service-Taste betätigen !'}		
{attribute 'Message.Info' := '%Var1'}
{attribute 'Message.Type' := '8'}	
{attribute 'Message.Log'  := '1'}
{attribute 'Message.Var1' := 'sBMK'}  	
	bMeldReset			:BOOL;	
	
	sBMK					:T_MaxString;
	
END_STRUCT
END_TYPE

// DUTs/HMI_Meldungen/Meldelisten/InternAchsen/ST_MeldAchsGruppe
{attribute 'pack_mode' := '1'}
TYPE ST_MeldAchsGruppe :
STRUCT
{attribute 'Message.SourceID'}
	SourceID			:DINT;
	
{attribute 'Message.SourceName'}
   SourceName		:STRING	:= 'Achgruppen';

	
{attribute 'Message.Text' := 'Achsgruppenfehler: %Var2'}		
{attribute 'Message.Info' := '%Var1'}
{attribute 'Message.Type' := '8'}	
{attribute 'Message.Log'  := '1'}
{attribute 'Message.Var1' := 'sBMK'}  	
{attribute 'Message.Var2' := 'sText'}
	bMeldFehler		:BOOL;	
	
	sText				:T_MaxString;
	sBMK				:T_MaxString;
END_STRUCT
END_TYPE

// DUTs/HMI_Meldungen/Meldelisten/InternEinspeis/ST_MeldAuffrischKlemme
{attribute 'pack_mode' := '1'}
TYPE ST_MeldAuffrischKlemme :
STRUCT
{attribute 'Message.SourceID'}
	SourceID					:DINT;
	
{attribute 'Message.SourceName'}
   SourceName				:STRING	:= 'Auffrischungsklemme';

{attribute 'Message.Text' := 'Auffrischungsklemme meldet Us-Unterspannung (Einspeisung)! (%Var1)'}
{attribute 'Message.Info' := '%Var1'}
{attribute 'Message.Type' := '8'}	
{attribute 'Message.Log'  := '1'}
{attribute 'Message.Var1' := 'sBMK'}  	
	bMeldUnterspannung		:BOOL;	// Zu kleine Spannung/Unterspannung an einer EL9110 oder so
{attribute 'Message.Text' := 'Auffrischungsklemme meldet Up-Unterspannung (Power)! (%Var1)'}                                                             
{attribute 'Message.Info' := '%Var1'}
{attribute 'Message.Type' := '8'} 
{attribute 'Message.Log'  := '1'}
{attribute 'Message.Var1' := 'sBMK'}                        
	bMeldPowerUnterspannung	:BOOL;  // Spannung an den Powerkontakten
	
	sBMK							:T_MaxString;
END_STRUCT
END_TYPE

// DUTs/HMI_Meldungen/Meldelisten/InternEinspeis/ST_MeldEinspeisKlemme
{attribute 'pack_mode' := '1'}
TYPE ST_MeldEinspeisKlemme :
STRUCT
{attribute 'Message.SourceID'}
	SourceID				:DINT;
	
{attribute 'Message.SourceName'}
   SourceName			:STRING	:= 'Potenzialeinspeisung';

{attribute 'Message.Text' := 'Fehler Einspeisung für Ausgänge %Var2 erkannt ! (%Var1)'}		
{attribute 'Message.Info' := '%Var1'}
{attribute 'Message.Type' := '8'}	
{attribute 'Message.Log'  := '1'}
{attribute 'Message.Var1' := 'sBMK'}  		
{attribute 'Message.Var2' := 'sPotentialName'}
	bMeldEinspeis		:BOOL;	// Fehler durch zu spätes Ausschalten oder nicht eingeschaltet
{attribute 'Message.Text' := 'Fehler Rückeinspeisung für Ausgänge %Var2 erkannt ! (%Var1)'}		
{attribute 'Message.Info' := '%Var1'}
{attribute 'Message.Type' := '8'}	
{attribute 'Message.Log'  := '1'}
{attribute 'Message.Var1' := 'sBMK'}  		
{attribute 'Message.Var2' := 'sPotentialName'}  
	bMeldRueckspeis	:BOOL;	// Fehler durch Querschluss
	
	sBMK					:T_MaxString;
	sPotentialName		:T_MaxString;
END_STRUCT
END_TYPE

// DUTs/HMI_Meldungen/Meldelisten/InternSafety/ST_MeldKlemme
{attribute 'pack_mode' := '1'}
TYPE ST_MeldKlemme :
STRUCT
{attribute 'Message.SourceID'}
	SourceID			:DINT;
	
{attribute 'Message.SourceName'}
   SourceName		:STRING	:= 'Safety-Klemmen';

{attribute 'Message.Text' := '%Var1 (%Var2)'}		
{attribute 'Message.Info' := '%Var2'}
{attribute 'Message.Type' := '8'}	
{attribute 'Message.Log'  := '1'}
{attribute 'Message.Var1' := 'sMeld'}  		
{attribute 'Message.Var2' := 'sBMK'}
	bMeld				:BOOL;
	
	sMeld				:T_MaxString;
	sBMK				:T_MaxString;
	
END_STRUCT
END_TYPE

// DUTs/HMI_Meldungen/Meldelisten/InternSafety/ST_MeldSafetyFBErrors
{attribute 'pack_mode' := '1'}
TYPE ST_MeldSafetyFBErrors :
STRUCT
{attribute 'Message.SourceID'}
	SourceID			:DINT;
	
{attribute 'Message.SourceName'}
   SourceName		:STRING	:= 'TwinSAFE';

{attribute 'Message.Text' := '%Var1'}		
{attribute 'Message.Info' := ''}
{attribute 'Message.Type' := '8'}	
{attribute 'Message.Log'  := '1'}
{attribute 'Message.Var1' := 'sMeldFBError_ErrorState'}
	bMeldFBError_ErrorState		:BOOL;

{attribute 'Message.Text' := '%Var1'}		
{attribute 'Message.Info' := ''}
{attribute 'Message.Type' := '8'}	
{attribute 'Message.Log'  := '1'}
{attribute 'Message.Var1' := 'sMeldFBError_ErrorDiag'}
	bMeldFBError_ErrorDiag		:BOOL;
	
	sMeldFBError_ErrorState		:T_MaxString;
	sMeldFBError_ErrorDiag		:T_MaxString;
	
END_STRUCT
END_TYPE

// DUTs/HMI_Meldungen/Meldelisten/InternSafety/ST_MeldSafetygruppe
{attribute 'pack_mode' := '1'}
TYPE ST_MeldSafetygruppe :
STRUCT
{attribute 'Message.SourceID'}
	SourceID					:DINT;
	
{attribute 'Message.SourceName'}
   SourceName				:STRING	:= 'TwinSAFE';
 
{attribute 'Message.Text' := '%Var1'}		
{attribute 'Message.Info' := ''}
{attribute 'Message.Type' := '8'}	
{attribute 'Message.Log'  := '1'}
{attribute 'Message.Var1' := 'sGruppe'}  
	bMeldAusg				:BOOL;
	
{attribute 'Message.Text' := '%Var1'}		
{attribute 'Message.Info' := ''}
{attribute 'Message.Type' := '8'}	
{attribute 'Message.Log'  := '1'}
{attribute 'Message.Var1' := 'sMeldFBErrorGruppe'}
	bMeldFBErrorGrp		:BOOL;

	sGruppe					:T_MaxString;
	sMeldFBErrorGruppe	:T_MaxString;
END_STRUCT
END_TYPE

// DUTs/HMI_Meldungen/Meldelisten/InternSafety/ST_MeldSafetyOuts
{attribute 'pack_mode' := '1'}
TYPE ST_MeldSafetyOuts :
STRUCT
{attribute 'Message.SourceID'}
	SourceID			:DINT;
	
{attribute 'Message.SourceName'}
   SourceName		:STRING	:= 'TwinSAFE';
	
{attribute 'Message.Text' := '%Var1 (%Var2)'}		
{attribute 'Message.Info' := '%Var2'}
{attribute 'Message.Type' := '8'}	
{attribute 'Message.Log'  := '1'}
{attribute 'Message.Var1' := 'sDiag'}
{attribute 'Message.Var2' := 'sBMK'}
	bMeldDiag		:BOOL;
	
{attribute 'Message.Text' := '%Var1 (%Var2)'}		
{attribute 'Message.Info' := '%Var2'}
{attribute 'Message.Type' := '8'}	
{attribute 'Message.Log'  := '1'}
{attribute 'Message.Var1' := 'sState'}
{attribute 'Message.Var2' := 'sBMK'}
	bMeldState		:BOOL;
	
	sDiag				:T_MaxString;
	sState			:T_MaxString;
	sBMK				:T_MaxString;
	
END_STRUCT
END_TYPE

// DUTs/HMI_Meldungen/Meldelisten/InternSchaltschrank/ST_MeldElektrSichg
{attribute 'pack_mode' := '1'}
TYPE ST_MeldElektrSichg :
STRUCT
	 
{attribute 'Message.SourceID'}
	SourceID		:DINT;
	
{attribute 'Message.SourceName'}
   SourceName	:STRING	:= 'Schaltschrank';
 
{attribute 'Message.Text' := 'Elektronische Sicherung: %Var2 (%Var1)'}		
{attribute 'Message.Info' := '%Var1'}
{attribute 'Message.Type' := '8'}	
{attribute 'Message.Log'  := '1'}
{attribute 'Message.Var1' := 'sBMK'}  
{attribute 'Message.Var2' := 'sText'}  
	bMeldAusg	:BOOL;

	sBMK			:T_MaxString;
	sText			:T_MaxString;
	
END_STRUCT
END_TYPE

// DUTs/HMI_Meldungen/Meldelisten/InternSchaltschrank/ST_MeldKlimaGeraet
{attribute 'pack_mode' := '1'}
TYPE ST_MeldKlimaGeraet :
STRUCT
	 
{attribute 'Message.SourceID'}
	SourceID		:DINT;
	
{attribute 'Message.SourceName'}
   SourceName	:STRING	:= 'Schaltschrank';
 
{attribute 'Message.Text' := 'Klimagerät meldet nicht betriebsbereit oder Schaltschranktür offen ! (%Var1)'}		
{attribute 'Message.Info' := '%Var1'}
{attribute 'Message.Type' := '1'}	
{attribute 'Message.Log'  := '0'}
{attribute 'Message.Var1' := 'sBMK'}  
	bMeldAusg	:BOOL;

	sBMK			:T_MaxString;

END_STRUCT
END_TYPE

// DUTs/HMI_Meldungen/Meldelisten/InternSchaltschrank/ST_MeldMotSchutzS
{attribute 'pack_mode' := '1'}
TYPE ST_MeldMotSchutzS :
STRUCT
	 
{attribute 'Message.SourceID'}
	SourceID		:DINT;
	
{attribute 'Message.SourceName'}
   SourceName	:STRING	:= 'Schaltschrank';
 
{attribute 'Message.Text' := 'Motorschutzschalter hat ausgelöst ! (%Var1)'}		
{attribute 'Message.Info' := '%Var1'}
{attribute 'Message.Type' := '8'}	
{attribute 'Message.Log'  := '1'}
{attribute 'Message.Var1' := 'sBMK'}  
	bMeldAusg	:BOOL;	

	sBMK			:T_MaxString;
	
END_STRUCT
END_TYPE

// DUTs/HMI_Meldungen/Meldelisten/InternSchaltschrank/ST_MeldSchaltNetzT
{attribute 'pack_mode' := '1'}
TYPE ST_MeldSchaltNetzT :
STRUCT
	 
{attribute 'Message.SourceID'}
	SourceID		:DINT;
	
{attribute 'Message.SourceName'}
   SourceName	:STRING	:= 'Schaltschrank';
 
{attribute 'Message.Text' := '24V-Netzteil meldet(e) Unterspannung ! (%Var1)'}		
{attribute 'Message.Info' := '%Var1'}
{attribute 'Message.Type' := '8'}	
{attribute 'Message.Log'  := '1'}
{attribute 'Message.Var1' := 'sBMK'}  
	bMeldAusg	:BOOL;	

	sBMK			:T_MaxString;
	
END_STRUCT
END_TYPE

// DUTs/HMI_Meldungen/Meldelisten/InternSchaltschrank/ST_MeldSichgAutom
{attribute 'pack_mode' := '1'}
TYPE ST_MeldSichgAutom :
STRUCT
	 
{attribute 'Message.SourceID'}
	SourceID		:DINT;
	
{attribute 'Message.SourceName'}
   SourceName	:STRING	:= 'Schaltschrank';
 
{attribute 'Message.Text' := 'Sicherungsautomat hat ausgelöst ! (%Var1)'}		
{attribute 'Message.Info' := '%Var1'}
{attribute 'Message.Type' := '8'}	
{attribute 'Message.Log'  := '1'}
{attribute 'Message.Var1' := 'sBMK'}  
	bMeldAusg	:BOOL;	

	sBMK			:T_MaxString;
	
END_STRUCT
END_TYPE

// DUTs/HMI_Meldungen/Meldelisten/InternSchaltschrank/ST_MeldThermoUeberw
{attribute 'pack_mode' := '1'}
TYPE ST_MeldThermoUeberw :
STRUCT
	 
{attribute 'Message.SourceID'}
	SourceID		:DINT;
	
{attribute 'Message.SourceName'}
   SourceName	:STRING	:= 'Schaltschrank';
 
{attribute 'Message.Text' := 'Thermoüberwachung hat ausgelöst ! (%Var1)'}		
{attribute 'Message.Info' := '%Var1'}
{attribute 'Message.Type' := '8'}	
{attribute 'Message.Log'  := '1'}
{attribute 'Message.Var1' := 'sBMK'}  
	bMeldAusg	:BOOL;	

	sBMK			:T_MaxString;
	
END_STRUCT
END_TYPE

// DUTs/HMI_Meldungen/Meldelisten/InternSchaltschrank/ST_MeldUSV
{attribute 'pack_mode' := '1'}
TYPE ST_MeldUSV :
STRUCT	 
{attribute 'Message.SourceID'}
	SourceID			:DINT;
	
{attribute 'Message.SourceName'}
   SourceName		:STRING	:= 'Schaltschrank';
 
{attribute 'Message.Text' := 'Bitte wechseln Sie die Batterie der USV aus ! (%Var1)'}		
{attribute 'Message.Info' := '%Var1'}
{attribute 'Message.Type' := '1'}	
{attribute 'Message.Log'  := '1'}
{attribute 'Message.Var1' := 'sBMK'}  
	bMeldAustausch		:BOOL;	

{attribute 'Message.Text' := 'USV - Status unbekannt !(%Var1)'}		
{attribute 'Message.Info' := '%Var1'}
{attribute 'Message.Type' := '1'}	
{attribute 'Message.Log'  := '1'}
{attribute 'Message.Var1' := 'sBMK'}  
	bMeldStatusUnbekannt	:BOOL;	

{attribute 'Message.Text' := 'Fehler in der Kommunikation zur USV ! (%Var1)'}		
{attribute 'Message.Info' := '%Var1'}
{attribute 'Message.Type' := '1'}	
{attribute 'Message.Log'  := '1'}
{attribute 'Message.Var1' := 'sBMK'}  
	bMeldKommFehler		:BOOL;	

{attribute 'Message.Text' := 'USV auf Batteriebetrieb ! (%Var1)'}		
{attribute 'Message.Info' := '%Var1'}
{attribute 'Message.Type' := '1'}	
{attribute 'Message.Log'  := '1'}
{attribute 'Message.Var1' := 'sBMK'}  
	bMeldBatteriebetrieb	:BOOL;	

{attribute 'Message.Text' := 'USV - Batterie am unteren Level ! (%Var1)'}		
{attribute 'Message.Info' := '%Var1'}
{attribute 'Message.Type' := '7'}	
{attribute 'Message.Log'  := '1'}
{attribute 'Message.Var1' := 'sBMK'}  
	bMeldUnteresLevel		:BOOL;	

{attribute 'Message.Text' := 'USV - Batterie am kritischen Level ! (%Var1)'}		
{attribute 'Message.Info' := '%Var1'}
{attribute 'Message.Type' := '7'}	
{attribute 'Message.Log'  := '1'}
{attribute 'Message.Var1' := 'sBMK'}  
	bMeldKritLevel		:BOOL;	

	sBMK					:T_MaxString;

END_STRUCT
END_TYPE

// DUTs/HMI_Meldungen/Meldelisten/InternSchutzbereich/ST_MeldNotHalt
{attribute 'pack_mode' := '1'}
TYPE ST_MeldNotHalt :
STRUCT
{attribute 'Message.SourceID'}
	SourceID			:DINT;

{attribute 'Message.SourceName'}
   SourceName		:STRING	:= 'Sicherheitseinrichtung';

{attribute 'Message.Text' := 'Not-Halt %Var2 wurde/ist betätigt ! (%Var1)'}
{attribute 'Message.Info' := '%Var1'}
{attribute 'Message.Type' := '8'}
{attribute 'Message.Log'  := '1'}
{attribute 'Message.Var1' := 'sBMK'}
{attribute 'Message.Var2' := 'sAktorName'}
	bMeldAusg		:BOOL;
{attribute 'Message.Text' := 'Not-Halt %Var2 war betätigt und kann quittiert werden ! (%Var1)'}
{attribute 'Message.Info' := '%Var1'}
{attribute 'Message.Type' := '4'}
{attribute 'Message.Log'  := '1'}
{attribute 'Message.Var1' := 'sBMK'}
{attribute 'Message.Var2' := 'sAktorName'}
	bMeldWarBetaetigt	:BOOL;	

	sAktorName		:T_MaxString;
	sBMK				:T_MaxString;
	
END_STRUCT
END_TYPE

// DUTs/HMI_Meldungen/Meldelisten/InternSchutzbereich/ST_MeldSchutzbereichOffen
{attribute 'pack_mode' := '1'}
TYPE ST_MeldSchutzbereichOffen :
STRUCT
	 
{attribute 'Message.SourceID'}
	SourceID			:DINT;
	
{attribute 'Message.SourceName'}
   SourceName		:STRING	:= 'Schutzbereiche';
 
{attribute 'Message.Text' := 'Schutzbereich unterbrochen -> Türen prüfen'}	
{attribute 'Message.Info' := ''}
{attribute 'Message.Type' := '4'}	
{attribute 'Message.Log'  := '1'} 
	bMeldUnterbrochen		:BOOL;
	
END_STRUCT
END_TYPE

// DUTs/HMI_Meldungen/Meldelisten/InternSchutzbereich/ST_MeldSichLichtg
{attribute 'pack_mode' := '1'}
TYPE ST_MeldSichLichtg :
STRUCT
	 
{attribute 'Message.SourceID'}
	SourceID			:DINT;
	
{attribute 'Message.SourceName'}
   SourceName		:STRING	:= 'Schutzbereiche';
 
{attribute 'Message.Text' := 'Lichtschutzgitter %Var1 unterbrochen / nicht quittiert ! (%Var2)'}	
{attribute 'Message.Info' := '%Var1'}
{attribute 'Message.Type' := '4'}	
{attribute 'Message.Log'  := '1'}
{attribute 'Message.Var1' := 'sAktorName'}  
{attribute 'Message.Var2' := 'sBMK'}  
	bMeldAusg		:BOOL;	

	sAktorName		:T_MaxString;
	sBMK				:T_MaxString;

END_STRUCT
END_TYPE

// DUTs/HMI_Meldungen/Meldelisten/InternSchutzbereich/ST_MeldStHLuft
{attribute 'pack_mode' := '1'}
TYPE ST_MeldStHLuft :
STRUCT
	 
{attribute 'Message.SourceID'}
	SourceID			:DINT;
	
{attribute 'Message.SourceName'}
   SourceName		:STRING	:= 'Schutzbereich';
 
{attribute 'Message.Text' := 'Betriebsdruck Steuerhilfsluft ist nicht abgebaut ! (%Var1)'}	
{attribute 'Message.Info' := '%Var1'}
{attribute 'Message.Type' := '4'}	
{attribute 'Message.Log'  := '1'}
{attribute 'Message.Var1' := 'sBMK1'}  
	bMeldNichtAbgebaut		:BOOL;	

{attribute 'Message.Text' := 'Betriebsdruck Steuerhilfsluft ist nicht aufgebaut ! (%Var1)'}	
{attribute 'Message.Info' := '%Var1'}
{attribute 'Message.Type' := '4'}	
{attribute 'Message.Log'  := '1'}
{attribute 'Message.Var1' := 'sBMK2'}  
	bMeldNichtAufgebaut		:BOOL;	

{attribute 'Message.Text' := 'Automatikbetrieb gesperrt, da Steuerhilfsluft überbrückt ! (%Var1)'}	
{attribute 'Message.Info' := '%Var1'}
{attribute 'Message.Type' := '1'}	
{attribute 'Message.Log'  := '1'}
{attribute 'Message.Var1' := 'sBMK2'}  
	bMeldUeberbrueckt			:BOOL;	

{attribute 'Message.Text' := 'Schlüsselschalter Steuerhilfsluft betätigt, aber Schutzbereich nicht geschlossen. Steuerhilfsluft wird nicht freigegeben! (%Var1)'}	
{attribute 'Message.Info' := '%Var1'}
{attribute 'Message.Type' := '1'}	
{attribute 'Message.Log'  := '1'}
{attribute 'Message.Var1' := 'sBMK2'}  
	bMeldNichtFreigegeben	:BOOL;

	sBMK1				:T_MaxString;	// Sensor 1
	sBMK2				:T_MaxString;	// Sensor 2
	
END_STRUCT
END_TYPE

// DUTs/HMI_Meldungen/Meldelisten/InternSchutzbereich/ST_MeldTuerFrgBremsentest
{attribute 'pack_mode' := '1'}
TYPE ST_MeldTuerFrgBremsentest :
STRUCT
{attribute 'Message.SourceID'}
	SourceID			:DINT;
	
{attribute 'Message.SourceName'}
   SourceName		:STRING	:= 'Schutzbereiche';
	
{attribute 'Message.Text' := 'Schutztüren durch fehlerhaften Bremsentest gesperrt ! '}		
{attribute 'Message.Info' := ''}
{attribute 'Message.Type' := '4'}	
{attribute 'Message.Log'  := '1'}
	bMeldGesperrt	:BOOL;	

	
END_STRUCT
END_TYPE

// DUTs/HMI_Meldungen/Meldelisten/InternSchutzbereich/ST_MeldWartgTuer
{attribute 'pack_mode' := '1'}
TYPE ST_MeldWartgTuer :
STRUCT
	 
{attribute 'Message.SourceID'}
	SourceID			:DINT;
	
{attribute 'Message.SourceName'}
   SourceName		:STRING	:= 'Schutzbereiche';
 
{attribute 'Message.Text' := '%Var2 ist geöffnet/nicht quittiert ! (%Var1)'}	
{attribute 'Message.Info' := '%Var1'}
{attribute 'Message.Type' := '4'}	
{attribute 'Message.Log'  := '1'} 
{attribute 'Message.Var1' := 'sBMK'} 
{attribute 'Message.Var2' := 'sAktorName'}  
	bMeldGeoeffnet		:BOOL;	

{attribute 'Message.Text' := 'Automatik Halt %Var2 ist aktiv ! (%Var1)'}	
{attribute 'Message.Info' := '%Var1'}
{attribute 'Message.Type' := '1'}	
{attribute 'Message.Log'  := '1'}
{attribute 'Message.Var1' := 'sBMK'}  
{attribute 'Message.Var2' := 'sAktorName'}  
	bMeldAutoHalt		:BOOL;	

{attribute 'Message.Text' := '%Var2 ist angewählt ! (%Var1)'}	
{attribute 'Message.Info' := '%Var1'}
{attribute 'Message.Type' := '1'}	
{attribute 'Message.Log'  := '1'}
{attribute 'Message.Var1' := 'sBMK'}  
{attribute 'Message.Var2' := 'sAktorName'}  
	bMeldAnwahl			:BOOL;	// Meldung für Schutztür ist angewählt. Vorallem gedacht für die Schutztüranwahl von einem anderen Steuerungsbereich

	sAktorName		:T_MaxString;
	sBMK				:T_MaxString;
	
END_STRUCT
END_TYPE

// DUTs/HMI_Meldungen/Meldelisten/InternSonstiges/ST_MeldADS_ExchangeError
{attribute 'pack_mode' := '1'}
TYPE ST_MeldADS_ExchangeError :
STRUCT
{attribute 'Message.SourceID'}
	SourceID			:DINT;
	
{attribute 'Message.SourceName'}
   SourceName		:STRING	:= 'ADS-Kommunikation';
	
{attribute 'Message.Text' := 'ADS-Exchange: %Var1'}	
{attribute 'Message.Info' := ''}
{attribute 'Message.Type' := '1'}	
{attribute 'Message.Log'  := '1'}
{attribute 'Message.Var1' := 'sError'}
	bError			:BOOL;
	sError			:T_MaxString;
	
END_STRUCT
END_TYPE

// DUTs/HMI_Meldungen/Meldelisten/InternSonstiges/ST_MeldADSKommError
{attribute 'pack_mode' := '1'}
TYPE ST_MeldADSKommError :
STRUCT
{attribute 'Message.SourceID'}
	SourceID			:DINT;
	
{attribute 'Message.SourceName'}
   SourceName		:STRING	:= 'ADS-Kommunikation';
	
{attribute 'Message.Text' := 'Signalkommunikation: Keine Kommunikation mit der %Var1 vorhanden!!'}		
{attribute 'Message.Info' := ''}
{attribute 'Message.Type' := '1'}	
{attribute 'Message.Log'  := '1'}
{attribute 'Message.Var1'  := 'sAnlagenteil'}
	bMeldKommError		:BOOL;	
	sAnlagenteil		:T_MaxString;	
	
END_STRUCT
END_TYPE

// DUTs/HMI_Meldungen/Meldelisten/InternSonstiges/ST_MeldBetriebsdruck
{attribute 'pack_mode' := '1'}
TYPE ST_MeldBetriebsdruck :
STRUCT
{attribute 'Message.SourceID'}
	SourceID			:DINT;
	
{attribute 'Message.SourceName'}
   SourceName		:STRING	:= 'Anlage Allgemein';
	
{attribute 'Message.Text' := 'Betriebsdruck nicht aufgebaut oder unterschritten ! Bitte Druckluftversorgung überprüfen ! (%Var1)'}		
{attribute 'Message.Info' := '%Var1'}
{attribute 'Message.Type' := '7'}	
{attribute 'Message.Log'  := '1'}
{attribute 'Message.Var1' := 'sBMK'}
	bMeldBetriebsdruck	:BOOL;	// Betriebsdruck nicht aufgebaut
	
{attribute 'Message.Text' := 'Betriebsdruck ist abgeschaltet! Wird mit Steuerung EIN wieder eingeschaltet! (%Var1)'}		
{attribute 'Message.Info' := '%Var1'}
{attribute 'Message.Type' := '1'}	
{attribute 'Message.Log'  := '1'}
{attribute 'Message.Var1' := 'sBMK'}
	bMeldAbgeschaltet	:BOOL;	// Betriebsdruck nicht aufgebaut
	
	sBMK				:T_MaxString;

	
END_STRUCT
END_TYPE

// DUTs/HMI_Meldungen/Meldelisten/InternSonstiges/ST_MeldDatenanf
{attribute 'pack_mode' := '1'}
TYPE ST_MeldDatenanf :
STRUCT
{attribute 'Message.SourceID'}
	SourceID			:DINT;
	
{attribute 'Message.SourceName'}
   SourceName		:STRING	:= 'Datenanforderung';
	
{attribute 'Message.Text' := 'Neuanforderung mit Hinweistaste! (Automatik Aus!) (Step: %Var1)'}		
{attribute 'Message.Info' := ''}
{attribute 'Message.Type' := '1'}	
{attribute 'Message.Log'  := '1'}
{attribute 'Message.Var1' := 'sStepInfo'}
	bMeldAnfFehler		:BOOL;
	
	sStepInfo		:T_MaxString;	

END_STRUCT
END_TYPE

// DUTs/HMI_Meldungen/Meldelisten/InternSonstiges/ST_MeldEAPKommError
{attribute 'pack_mode' := '1'}
TYPE ST_MeldEAPKommError :
STRUCT
{attribute 'Message.SourceID'}
	SourceID			:DINT;
	
{attribute 'Message.SourceName'}
   SourceName		:STRING	:= 'EAP-Kommunikation';
	
{attribute 'Message.Text' := 'Kommunikation mit %Var1: Keine Kommunikation vorhanden!'}	
{attribute 'Message.Info' := ''}
{attribute 'Message.Type' := '1'}	
{attribute 'Message.Log'  := '1'}
{attribute 'Message.Var1' := 'sAnlagenteil'}
	bMeldKommError			:BOOL;

{attribute 'Message.Text' := 'Kommunikation mit %Var1: Signalstärke schwach, Leitung prüfen!'}	
{attribute 'Message.Info' := ''}
{attribute 'Message.Type' := '1'}	
{attribute 'Message.Log'  := '1'}
{attribute 'Message.Var1' := 'sAnlagenteil'}
	bMeldKeinSignal		:BOOL;
	
{attribute 'Message.Text' := 'Kommunikation mit %Var1: Ethernetframe wird nicht gesendet!'}	
{attribute 'Message.Info' := ''}
{attribute 'Message.Type' := '1'}	
{attribute 'Message.Log'  := '1'}
{attribute 'Message.Var1' := 'sAnlagenteil'}
	bMeldNichtSendebereit		:BOOL;

{attribute 'Message.Text' := 'Kommunikation mit %Var1: Falsche ID(%Var2) zurückgemeldet! Bitte korrekte Reihenfolge in Datenpuffern kontrollieren und Hinweistaste betätigen!'}	
{attribute 'Message.Info' := ''}
{attribute 'Message.Type' := '1'}	
{attribute 'Message.Log'  := '1'}
{attribute 'Message.Var1' := 'sAnlagenteil'}
{attribute 'Message.Var2' := 'sErrorID'}
	bMeldFalscheID			:BOOL;

{attribute 'Message.Text' := 'Kommunikation mit %Var1: Zugehörige TwinSAFE Gruppe in Störung. Mögliche Ursachen sind: Partner PC ausgeschaltet, falsch konfiguriert, oder keine Netzwerkverbindung.'}	
{attribute 'Message.Info' := ''}
{attribute 'Message.Type' := '1'}	
{attribute 'Message.Log'  := '1'}
{attribute 'Message.Var1' := 'sAnlagenteil'}
	bMeldTwinSafeGrp		:BOOL;

{attribute 'Message.Text' := 'Kommunikation mit %Var1: Unbekannter TwinSAFE Fehler!'}	
{attribute 'Message.Info' := ''}
{attribute 'Message.Type' := '1'}	
{attribute 'Message.Log'  := '1'}
{attribute 'Message.Var1' := 'sAnlagenteil'}
	bMeldTwinSafeFehler	:BOOL;

{attribute 'Message.Text' := 'Kommunikation mit %Var1: Zugehörige TwinSAFE Connection Info im ungültigen Zustand!'}	
{attribute 'Message.Info' := ''}
{attribute 'Message.Type' := '1'}	
{attribute 'Message.Log'  := '1'}
{attribute 'Message.Var1' := 'sAnlagenteil'}
	bMeldTwinSafeUngueltig	:BOOL;

	sAnlagenteil	:T_MaxString;
	sErrorID			:T_MaxString;
	
END_STRUCT
END_TYPE

// DUTs/HMI_Meldungen/Meldelisten/InternSonstiges/ST_MeldEtherCAT
{attribute 'pack_mode' := '1'}
TYPE ST_MeldEtherCAT :
STRUCT
{attribute 'Message.SourceID'}
	SourceID			:DINT;
	
{attribute 'Message.SourceName'}
   SourceName		:STRING	:= 'EtherCAT-Bus';
	
{attribute 'Message.Text' := 'EtherCAT Fehler !'}		
{attribute 'Message.Info' := ''}
{attribute 'Message.Type' := '8'}	
{attribute 'Message.Log'  := '1'}
	bMeldEtherCATFehler		:BOOL;	

{attribute 'Message.Text' := 'Anzahl der EtherCAT Slaves nicht korrekt !'}		
{attribute 'Message.Info' := ''}
{attribute 'Message.Type' := '8'}	
{attribute 'Message.Log'  := '1'}
	bMeldAnzSlavesFehler		:BOOL;

{attribute 'Message.Text' := '%Var1'}		
{attribute 'Message.Info' := ''}
{attribute 'Message.Type' := '8'}	
{attribute 'Message.Log'  := '1'}
{attribute 'Message.Var1' := 'sText'}  
	bMeldSlaveError			:BOOL;
	
	sText		:T_MaxString;

END_STRUCT
END_TYPE

// DUTs/HMI_Meldungen/Meldelisten/InternSonstiges/ST_MeldGrundstellung
{attribute 'pack_mode' := '1'}
TYPE ST_MeldGrundstellung :
STRUCT
	 
{attribute 'Message.SourceID'}
	SourceID			:DINT;
	
{attribute 'Message.SourceName'}
   SourceName		:STRING	:= 'Grundstellungsablauf';
 
{attribute 'Message.Text' := 'Grundstellung wird ausgeführt /bitte warten !'}		
{attribute 'Message.Info' := ''}
{attribute 'Message.Type' := '1'}	
{attribute 'Message.Log'  := '1'}
	bMeldAktiv	:BOOL;	

{attribute 'Message.Text' := 'Grundstellung wurde ausgeführt /bitte Teil(e) entnehmen !'}	
{attribute 'Message.Info' := ''}
{attribute 'Message.Type' := '1'}	
{attribute 'Message.Log'  := '1'}
	bMeldDonemitEntnahme	:BOOL;

{attribute 'Message.Text' := 'Grundstellung wurde ausgeführt !'}	
{attribute 'Message.Info' := ''}
{attribute 'Message.Type' := '1'}	
{attribute 'Message.Log'  := '1'}
	bMeldDoneOhneEntnahme	:BOOL;

END_STRUCT
END_TYPE

// DUTs/HMI_Meldungen/Meldelisten/InternSonstiges/ST_MeldIOLinkKlemme
{attribute 'pack_mode' := '1'}
TYPE ST_MeldIOLinkKlemme :
STRUCT
{attribute 'Message.SourceID'}
	SourceID			:DINT;
	
{attribute 'Message.SourceName'}
   SourceName		:STRING	:= 'EtherCAT-Bus';

{attribute 'Message.Text' := 'IO-Link Fehler: %Var1'}		
{attribute 'Message.Info' := '%Var2'}
{attribute 'Message.Type' := '8'}	
{attribute 'Message.Log'  := '1'}
{attribute 'Message.Var1' := 'sText1'}
{attribute 'Message.Var2' := 'sBMK1'}
	bMeld1		:BOOL;
{attribute 'Message.Text' := 'IO-Link Fehler: %Var1'}		
{attribute 'Message.Info' := '%Var2'}
{attribute 'Message.Type' := '8'}	
{attribute 'Message.Log'  := '1'}
{attribute 'Message.Var1' := 'sText2'}
{attribute 'Message.Var2' := 'sBMK2'}
	bMeld2		:BOOL;
{attribute 'Message.Text' := 'IO-Link Fehler: %Var1'}		
{attribute 'Message.Info' := '%Var2'}
{attribute 'Message.Type' := '8'}	
{attribute 'Message.Log'  := '1'}
{attribute 'Message.Var1' := 'sText3'}
{attribute 'Message.Var2' := 'sBMK3'}
	bMeld3		:BOOL;
{attribute 'Message.Text' := 'IO-Link Fehler: %Var1'}		
{attribute 'Message.Info' := '%Var2'}
{attribute 'Message.Type' := '8'}	
{attribute 'Message.Log'  := '1'}
{attribute 'Message.Var1' := 'sText4'}
{attribute 'Message.Var2' := 'sBMK4'}
	bMeld4		:BOOL;
	
	sText1		:STRING;
	sText2		:STRING;
	sText3		:STRING;
	sText4		:STRING;
	
	sBMK1			:T_MaxString;	// IO-Link Eingang 1
	sBMK2			:T_MaxString;	// IO-Link Eingang 2
	sBMK3			:T_MaxString;	// IO-Link Eingang 3
	sBMK4			:T_MaxString;	// IO-Link Eingang 4
END_STRUCT
END_TYPE

// DUTs/HMI_Meldungen/Meldelisten/UniAnstg/ST_MeldAchsKontrl
{attribute 'pack_mode' := '1'}
// Meldestruktur für Achsfehler an einer Achse aus dem FB_AchsKontrlAnstg
TYPE ST_MeldAchsKontrl :
STRUCT
	 
{attribute 'Message.SourceID'}
	SourceID			:DINT;
	
{attribute 'Message.SourceName'}
   SourceName		:STRING	:= 'Schaltschrank';
 
{attribute 'Message.Text' := 'Axis %Var1: %Var2 NC-Fehler ist aufgetreten ! (%Var3)'}
{attribute 'Message.Info' := '%Var3'}
{attribute 'Message.Type' := '8'}
{attribute 'Message.Log'  := '1'}
{attribute 'Message.Var1' := 'sAktorIdNr'}
{attribute 'Message.Var2' := 'sAktorName'}
{attribute 'Message.Var3' := 'sBMK'}
	bMeldNCFehler	:BOOL;

{attribute 'Message.Text' := 'Axis %Var1: %Var2 Antrieb ist nicht Betriebsbereit ! (%Var3)'}
{attribute 'Message.Info' := '%Var3'}
{attribute 'Message.Type' := '8'}
{attribute 'Message.Log'  := '1'}
{attribute 'Message.Var1' := 'sAktorIdNr'}
{attribute 'Message.Var2' := 'sAktorName'}
{attribute 'Message.Var3' := 'sBMK'}
	bMeldNichtBtB	:BOOL;

{attribute 'Message.Text' := 'Axis %Var1: %Var2 Istposition liegt nicht im gültigen Bereich ! (%Var3)'}
{attribute 'Message.Info' := '%Var3'}
{attribute 'Message.Type' := '7'}
{attribute 'Message.Log'  := '1'}
{attribute 'Message.Var1' := 'sAktorIdNr'}  
{attribute 'Message.Var2' := 'sAktorName'}  
{attribute 'Message.Var3' := 'sBMK'}
	bMeldIstPosUngueltig	:BOOL;

{attribute 'Message.Text' := 'Axis %Var1: %Var2 Zielposition liegt ausserhalb Softendlagen ! (%Var3)'}
{attribute 'Message.Info' := '%Var3'}
{attribute 'Message.Type' := '7'}
{attribute 'Message.Log'  := '1'}
{attribute 'Message.Var1' := 'sAktorIdNr'}  
{attribute 'Message.Var2' := 'sAktorName'}  
{attribute 'Message.Var3' := 'sBMK'}
	bMeldZielPosUngueltig	:BOOL;	

{attribute 'Message.Text' := 'Axis %Var1: %Var2 Zielposition wird nicht erreicht (Laufzeitfehler) ! (%Var3)'}
{attribute 'Message.Info' := '%Var3'}
{attribute 'Message.Type' := '7'}
{attribute 'Message.Log'  := '1'}
{attribute 'Message.Var1' := 'sAktorIdNr'}  
{attribute 'Message.Var2' := 'sAktorName'}  
{attribute 'Message.Var3' := 'sBMK'}
	bMeldLaufzeitfehler	:BOOL;	

{attribute 'Message.Text' := 'Axis %Var1: %Var2 Sicherheitsendlage Neg. wurde angefahren ! (%Var3)'}
{attribute 'Message.Info' := '%Var3'}
{attribute 'Message.Type' := '8'}
{attribute 'Message.Log'  := '1'}
{attribute 'Message.Var1' := 'sAktorIdNr'}  
{attribute 'Message.Var2' := 'sAktorName'}  
{attribute 'Message.Var3' := 'sEndlgBMK0'}
	bMeldEndlNeg	:BOOL;	

{attribute 'Message.Text' := 'Axis %Var1: %Var2 Sicherheitsendlage Pos. wurde angefahren ! (%Var3)'}
{attribute 'Message.Info' := '%Var3'}
{attribute 'Message.Type' := '8'}
{attribute 'Message.Log'  := '1'}
{attribute 'Message.Var1' := 'sAktorIdNr'}
{attribute 'Message.Var2' := 'sAktorName'}  
{attribute 'Message.Var3' := 'sEndlgBMK1'}
	bMeldEndlPos	:BOOL;

{attribute 'Message.Text' := 'Axis %Var1: %Var2 %Var3 !'}
{attribute 'Message.Info' := '%Var3'}
{attribute 'Message.Type' := '4'}
{attribute 'Message.Log'  := '1'}
{attribute 'Message.Var1' := 'sAktorIdNr'}
{attribute 'Message.Var2' := 'sAktorName'}
{attribute 'Message.Var3' := 'sBremsInfo'}
	bMeldBremsentest	:BOOL;

	sAktorIdNr		:T_MaxString:= 'AktorIdNr';
	sAktorName		:T_MaxString:= 'AktorName';
	sEndlgBMK0		:T_MaxString:= 'EndlgBMK0';
	sEndlgBMK1		:T_MaxString:= 'EndlgBMK1';
	sBremsInfo		:T_MaxString:= 'BremsInfo';
	sBMK				:T_MaxString;
	
END_STRUCT
END_TYPE

// DUTs/HMI_Meldungen/Meldelisten/UniAnstg/ST_MeldTextUniAchs
{attribute 'pack_mode' := '1'}
TYPE ST_MeldTextUniAchs :
STRUCT
	 
{attribute 'Message.SourceID'}
	SourceID			:DINT;
	
{attribute 'Message.SourceName'}
   SourceName		:STRING	:= 'Schaltschrank';
 
{attribute 'Message.Text' := 'Hinweis: %Var1 %Var2'}	
{attribute 'Message.Info' := 'Fehlerhinweis ID: %Var3'}
{attribute 'Message.Type' := '7'}	
{attribute 'Message.Log'  := '1'}
{attribute 'Message.Var1' := 'sBMK'}  
{attribute 'Message.Var2' := 'sMeldText'}  
{attribute 'Message.Var3' := 'sInfoText'}
	bMeldHinweis	:BOOL;	

{attribute 'Message.Text' := 'Axis %Var3: %Var1 Servoregler meldet nicht Betriebsbereit ! (%Var2)'}	
{attribute 'Message.Info' := ''}
{attribute 'Message.Type' := '8'}	
{attribute 'Message.Log'  := '1'}
{attribute 'Message.Var1' := 'sAktorName'}  
{attribute 'Message.Var2' := 'sBMK'}
{attribute 'Message.Var3' := 'sAchsnummer'}
	bStatMeldAusg	:BOOL;	

	sAktorName		:T_MaxString 	:= 'AktorName';
	sMeldText		:T_MaxString	:= 'MeldText';
	sInfoText		:T_MaxString	:= 'InfoText';
	sBMK				:T_MaxString;
	sAchsnummer		:T_MaxString;

END_STRUCT
END_TYPE

// DUTs/HMI_Meldungen/Meldelisten/UniAnstg/ST_MeldTextUniAktr
{attribute 'pack_mode' := '1'}
TYPE ST_MeldTextUniAktr :
STRUCT
	 
{attribute 'Message.SourceID'}
	SourceID			:DINT;
	
{attribute 'Message.SourceName'}
   SourceName		:STRING;
 
{attribute 'Message.Text' := 'Hinweis: %Var2 (%Var1)'}	
{attribute 'Message.Info' := 'Fehlerhinweis ID: %Var3'}
{attribute 'Message.Type' := '7'}	
{attribute 'Message.Log'  := '1'}
{attribute 'Message.Var1' := 'sBMK'}  
{attribute 'Message.Var2' := 'sMeldText'}
{attribute 'Message.Var3' := 'sInfoText'}
	bMeldHinweis	:BOOL;

{attribute 'Message.Text' := 'Laufzeitmeldung: %Var1 ! (%Var2)'}	
{attribute 'Message.Info' := ''}
{attribute 'Message.Type' := '7'}	
{attribute 'Message.Log'  := '1'}
{attribute 'Message.Var1' := 'sAktorName'}  
{attribute 'Message.Var2' := 'sBMK'}  
	bLfzMeldAusg	:BOOL;	

	sMeldText		:T_MaxString:= 'MeldText';
	sInfoText		:T_MaxString:= 'InfoText';
	sAktorName		:T_MaxString:= 'AktorName';
	sBMK				:T_MaxString;

END_STRUCT
END_TYPE

// DUTs/HMI_Meldungen/Meldelisten/UniAnstg/ST_MeldTextUniAntr
{attribute 'pack_mode' := '1'}
TYPE ST_MeldTextUniAntr :
STRUCT
	 
{attribute 'Message.SourceID'}
	SourceID			:DINT;
	
{attribute 'Message.SourceName'}
   SourceName		:STRING;
 
{attribute 'Message.Text' := 'Hinweis: %Var2 (%Var1)'}	
{attribute 'Message.Info' := 'Fehlerhinweis ID: %Var3'}
{attribute 'Message.Type' := '7'}	
{attribute 'Message.Log'  := '1'} 
{attribute 'Message.Var1' := 'sBMK'}  
{attribute 'Message.Var2' := 'sMeldText'}  
{attribute 'Message.Var3' := 'sInfoText'}
	bMeldHinweis	:BOOL;	

 
{attribute 'Message.Text' := 'Umrichterfehler: %Var2 (%Var1)'}	
{attribute 'Message.Info' := 'Fehlerhinweis ID: %Var3'}
{attribute 'Message.Type' := '8'}	
{attribute 'Message.Log'  := '1'} 
{attribute 'Message.Var1' := 'sBMK'}  
{attribute 'Message.Var2' := 'sMeldUmrichterfehler'}  
{attribute 'Message.Var3' := 'sInfoText'}
	bMeldFehlercode		:BOOL;	

{attribute 'Message.Text' := 'Frequenzumrichter: %Var1 meldet nicht Betriebsbereit ! (%Var2)'}	
{attribute 'Message.Info' := ''}
{attribute 'Message.Type' := '8'}	
{attribute 'Message.Log'  := '1'}
{attribute 'Message.Var1' := 'sAktorName'}  
{attribute 'Message.Var2' := 'sBMK'}  
	bMeldNichtBtb	:BOOL;
	
{attribute 'Message.Text' := 'Frequenzumrichter: %Var1 ist im STOP ! Bitte über das Bedienteil im Schaltschrank auf RUN stellen. (%Var2)'}	
{attribute 'Message.Info' := ''}
{attribute 'Message.Type' := '8'}	
{attribute 'Message.Log'  := '1'}
{attribute 'Message.Var1' := 'sAktorName'}  
{attribute 'Message.Var2' := 'sBMK'}  
	bMeldUmrichterGesperrt	:BOOL;
	
{attribute 'Message.Text' := '%Var1 Erstinbetriebnahme: Einlaufzyklus aktiv ! (%Var2)'}	
{attribute 'Message.Info' := ''}
{attribute 'Message.Type' := '1'}	
{attribute 'Message.Log'  := '1'}
{attribute 'Message.Var1' := 'sAktorName'}  
{attribute 'Message.Var2' := 'sBMK'}  
	bMeldEinlZyklAktiv	:BOOL;	

{attribute 'Message.Text' := '%Var1 Erstinbetriebnahme: Einlaufzyklus beendet ! (%Var2)'}	
{attribute 'Message.Info' := ''}
{attribute 'Message.Type' := '1'}	
{attribute 'Message.Log'  := '1'}
{attribute 'Message.Var1' := 'sAktorName'}  
{attribute 'Message.Var2' := 'sBMK'}  
	bMeldEinlZyklBeendet	:BOOL;	

{attribute 'Message.Text' := '%Var1 Betriebshinweis: Warmlaufzyklus aktiv ! (%Var2)'}	
{attribute 'Message.Info' := ''}
{attribute 'Message.Type' := '1'}	
{attribute 'Message.Log'  := '1'}
{attribute 'Message.Var1' := 'sAktorName'}  
{attribute 'Message.Var2' := 'sBMK'}  
	bMeldWarmlaufZykl		:BOOL;
	
{attribute 'Message.Text' := '%Var1 Referenzfahrt gestartet !'}	
{attribute 'Message.Info' := ''}
{attribute 'Message.Type' := '1'}	
{attribute 'Message.Log'  := '1'}
{attribute 'Message.Var1' := 'sAktorName'}  
	bMeldReffahrtStart	:BOOL;	
	
{attribute 'Message.Text' := '%Var1 nicht referenziert ! Bitte Referenzfahrt starten !'}	
{attribute 'Message.Info' := ''}
{attribute 'Message.Type' := '7'}	
{attribute 'Message.Log'  := '1'}
{attribute 'Message.Var1' := 'sAktorName'}  
	bMeldNichtReferenz	:BOOL;
	
{attribute 'Message.Text' := '%Var1 Laufzeitmeldung! Antrieb erreicht die negative Endlage nicht'}	
{attribute 'Message.Info' := ''}
{attribute 'Message.Type' := '7'}	
{attribute 'Message.Log'  := '1'}
{attribute 'Message.Var1' := 'sAktorName'}  
	bMeldLaufzeit0	:BOOL;	
	
{attribute 'Message.Text' := '%Var1 Laufzeitmeldung! Antrieb erreicht die positive Endlage nicht'}	
{attribute 'Message.Info' := ''}
{attribute 'Message.Type' := '7'}	
{attribute 'Message.Log'  := '1'}
{attribute 'Message.Var1' := 'sAktorName'}  
	bMeldLaufzeit1	:BOOL;	

	sMeldText		:STRING:= 'MeldText';
	sInfoText		:STRING:= 'InfoText';
	sAktorName		:STRING:= 'AktorName';
	sMeldUmrichterfehler	: STRING;
	sBMK				:STRING;

END_STRUCT
END_TYPE

// DUTs/HMI_Meldungen/Meldelisten/UniAnstg/ST_MeldTextUniWkzg
{attribute 'pack_mode' := '1'}
TYPE ST_MeldTextUniWkzg :
STRUCT
	 
{attribute 'Message.SourceID'}
	SourceID			:DINT;
	
{attribute 'Message.SourceName'}
   SourceName		:STRING;
 
{attribute 'Message.Text' := 'Hinweis: %Var2 (%Var1)'}	
{attribute 'Message.Info' := 'Fehlerhinweis ID: %Var3'}
{attribute 'Message.Type' := '7'}	
{attribute 'Message.Log'  := '1'}
{attribute 'Message.Var1' := 'sBMK'}  
{attribute 'Message.Var2' := 'sMeldText'}  
{attribute 'Message.Var3' := 'sInfoText'}
	bMeldHinweis	:BOOL;

	sMeldText		:T_MaxString:= 'MeldText';
	sInfoText		:T_MaxString:= 'InfoText';
	sAktorName		:T_MaxString:= 'AktorName';
	sBMK				:T_MaxString;

END_STRUCT
END_TYPE

// DUTs/HMI_Meldungen/Meldelisten/UniAnstg/ST_MeldTextUniZyli
{attribute 'pack_mode' := '1'}
TYPE ST_MeldTextUniZyli :
STRUCT
	 
{attribute 'Message.SourceID'}
	SourceID			:DINT;
	
{attribute 'Message.SourceName'}
   SourceName		:STRING;
 
{attribute 'Message.Text' := 'Hinweis: %Var1 %Var2'}	
{attribute 'Message.Info' := 'Fehlerhinweis ID: %Var3'}
{attribute 'Message.Type' := '7'}	
{attribute 'Message.Log'  := '1'}
{attribute 'Message.Var1' := 'sAktorName'}
{attribute 'Message.Var2' := 'sMeldText'}  
{attribute 'Message.Var3' := 'sInfoText'}
	bMeldHinweis	:BOOL;

{attribute 'Message.Text' := '%Var1 %Var2 (%Var3)'}	
{attribute 'Message.Info' := '}
{attribute 'Message.Type' := '7'}	
{attribute 'Message.Log'  := '1'}
{attribute 'Message.Var1' := 'sAktorName'}
{attribute 'Message.Var2' := 'sLzFehlerDef0'}
{attribute 'Message.Var3' := 'sBMK0'}
	bLfzMeldAusgDef0	:BOOL;	
{attribute 'Message.Text' := '%Var1 %Var2 (%Var3)'}	
{attribute 'Message.Info' := '}
{attribute 'Message.Type' := '7'}	
{attribute 'Message.Log'  := '1'}
{attribute 'Message.Var1' := 'sAktorName'}
{attribute 'Message.Var2' := 'sLzFehlerDef1'}
{attribute 'Message.Var3' := 'sBMK1'}
	bLfzMeldAusgDef1	:BOOL;	
{attribute 'Message.Text' := 'Sensorfehler: %Var1 (%Var2/%Var3)'}	
{attribute 'Message.Info' := '}
{attribute 'Message.Type' := '8'}	
{attribute 'Message.Log'  := '1'}
{attribute 'Message.Var1' := 'sSensorFehlDef'}
{attribute 'Message.Var2' := 'sBMK0'}  
{attribute 'Message.Var3' := 'sBMK1'}  
	bMeldSensFehlDef	:BOOL;	

{attribute 'Message.Text' := '%Var1 ist nicht in Grundstlg. ! (%Var2)'}	
{attribute 'Message.Info' := '}
{attribute 'Message.Type' := '7'}	
{attribute 'Message.Log'  := '1'}
{attribute 'Message.Var1' := 'sAktorName'}  
{attribute 'Message.Var2' := 'sBMK0'}  
	bLfzMeldAusg01	:BOOL;	
{attribute 'Message.Text' := '%Var1 ist nicht in Arbeitstlg. ! (%Var2)'}	
{attribute 'Message.Info' := '}
{attribute 'Message.Type' := '7'}	
{attribute 'Message.Log'  := '1'}
{attribute 'Message.Var1' := 'sAktorName'}  
{attribute 'Message.Var2' := 'sBMK1'}  
	bLfzMeldAusg11	:BOOL;	
{attribute 'Message.Text' := 'Sensorfehler: %Var1 Grund-/Arbeitstlg. ! (%Var2/%Var3)'}	
{attribute 'Message.Info' := '}
{attribute 'Message.Type' := '8'}	
{attribute 'Message.Log'  := '1'}
{attribute 'Message.Var1' := 'sAktorName'}  
{attribute 'Message.Var2' := 'sBMK0'}  
{attribute 'Message.Var3' := 'sBMK1'}  
	bMeldSensFehl1	:BOOL;	

{attribute 'Message.Text' := '%Var1 hat nicht abgesenkt ! (%Var2)'}	
{attribute 'Message.Info' := '}
{attribute 'Message.Type' := '7'}	
{attribute 'Message.Log'  := '1'}
{attribute 'Message.Var1' := 'sAktorName'}  
{attribute 'Message.Var2' := 'sBMK0'}  
	bLfzMeldAusg02	:BOOL;	
{attribute 'Message.Text' := '%Var1 hat nicht angehoben ! (%Var2)'}	
{attribute 'Message.Info' := '}
{attribute 'Message.Type' := '7'}	
{attribute 'Message.Log'  := '1'}
{attribute 'Message.Var1' := 'sAktorName'}  
{attribute 'Message.Var2' := 'sBMK1'}  
	bLfzMeldAusg12	:BOOL;	
{attribute 'Message.Text' := 'Sensorfehler: %Var1 absenk-/anheben ! (%Var2/%Var3)'}	
{attribute 'Message.Info' := '}
{attribute 'Message.Type' := '8'}	
{attribute 'Message.Log'  := '1'}
{attribute 'Message.Var1' := 'sAktorName'}  
{attribute 'Message.Var2' := 'sBMK0'}  
{attribute 'Message.Var3' := 'sBMK1'}  
	bMeldSensFehl2	:BOOL;	

{attribute 'Message.Text' := '%Var1 ist nicht eingefahren ! (%Var2)'}	
{attribute 'Message.Info' := '}
{attribute 'Message.Type' := '7'}	
{attribute 'Message.Log'  := '1'}
{attribute 'Message.Var1' := 'sAktorName'}  
{attribute 'Message.Var2' := 'sBMK0'}  
	bLfzMeldAusg03	:BOOL;	
{attribute 'Message.Text' := '%Var1 ist nicht ausgefahren ! (%Var2)'}	
{attribute 'Message.Info' := '}
{attribute 'Message.Type' := '7'}	
{attribute 'Message.Log'  := '1'}
{attribute 'Message.Var1' := 'sAktorName'}  
{attribute 'Message.Var2' := 'sBMK1'}  
	bLfzMeldAusg13	:BOOL;	
{attribute 'Message.Text' := 'Sensorfehler: %Var1 ein-/ausfahren ! (%Var2/%Var3)'}	
{attribute 'Message.Info' := '}
{attribute 'Message.Type' := '8'}	
{attribute 'Message.Log'  := '1'}
{attribute 'Message.Var1' := 'sAktorName'}  
{attribute 'Message.Var2' := 'sBMK0'}  
{attribute 'Message.Var3' := 'sBMK1'}  
	bMeldSensFehl3	:BOOL;	

{attribute 'Message.Text' := '%Var1 ist nicht zurückgefahren ! (%Var2)'}
{attribute 'Message.Info' := '}
{attribute 'Message.Type' := '7'}	
{attribute 'Message.Log'  := '1'}
{attribute 'Message.Var1' := 'sAktorName'}  
{attribute 'Message.Var2' := 'sBMK0'}  
	bLfzMeldAusg04	:BOOL;	
{attribute 'Message.Text' := '%Var1 ist nicht vorgefahren ! (%Var2)'}	
{attribute 'Message.Info' := '}
{attribute 'Message.Type' := '7'}	
{attribute 'Message.Log'  := '1'}
{attribute 'Message.Var1' := 'sAktorName'}  
{attribute 'Message.Var2' := 'sBMK1'}  
	bLfzMeldAusg14	:BOOL;	
{attribute 'Message.Text' := 'Sensorfehler: %Var1 zur-/vorfahren ! (%Var2/%Var3)'}	
{attribute 'Message.Info' := '}
{attribute 'Message.Type' := '8'}	
{attribute 'Message.Log'  := '1'}
{attribute 'Message.Var1' := 'sAktorName'}  
{attribute 'Message.Var2' := 'sBMK0'}  
{attribute 'Message.Var3' := 'sBMK1'}  
	bMeldSensFehl4	:BOOL;	

{attribute 'Message.Text' := '%Var1 ist nicht eingesteuert ! (%Var2)'}	
{attribute 'Message.Info' := '}
{attribute 'Message.Type' := '7'}	
{attribute 'Message.Log'  := '1'}
{attribute 'Message.Var1' := 'sAktorName'}  
{attribute 'Message.Var2' := 'sBMK0'}  
	bLfzMeldAusg05	:BOOL;	
{attribute 'Message.Text' := '%Var1 ist nicht ausgesteuert ! (%Var2)'}	
{attribute 'Message.Info' := '}
{attribute 'Message.Type' := '7'}	
{attribute 'Message.Log'  := '1'}
{attribute 'Message.Var1' := 'sAktorName'}  
{attribute 'Message.Var2' := 'sBMK1'}  
	bLfzMeldAusg15	:BOOL;	
{attribute 'Message.Text' := 'Sensorfehler: %Var1 ein-/aussteuern ! (%Var2/%Var3)'}	
{attribute 'Message.Info' := '}
{attribute 'Message.Type' := '8'}	
{attribute 'Message.Log'  := '1'}
{attribute 'Message.Var1' := 'sAktorName'}  
{attribute 'Message.Var2' := 'sBMK0'}  
{attribute 'Message.Var3' := 'sBMK1'}  
	bMeldSensFehl5	:BOOL;	

{attribute 'Message.Text' := '%Var1 hat nicht gelöst ! (%Var2)'}		
{attribute 'Message.Info' := '}
{attribute 'Message.Type' := '7'}	
{attribute 'Message.Log'  := '1'}
{attribute 'Message.Var1' := 'sAktorName'}  
{attribute 'Message.Var2' := 'sBMK0'}  
	bLfzMeldAusg06	:BOOL;	
{attribute 'Message.Text' := '%Var1 hat nicht gespannt ! (%Var2)'}	
{attribute 'Message.Info' := '}
{attribute 'Message.Type' := '7'}	
{attribute 'Message.Log'  := '1'}
{attribute 'Message.Var1' := 'sAktorName'}  
{attribute 'Message.Var2' := 'sBMK1'}  
	bLfzMeldAusg16	:BOOL;	
{attribute 'Message.Text' := 'Sensorfehler: %Var1 lösen/spannen ! (%Var2/%Var3)'}
{attribute 'Message.Info' := '}
{attribute 'Message.Type' := '8'}	
{attribute 'Message.Log'  := '1'}
{attribute 'Message.Var1' := 'sAktorName'}  
{attribute 'Message.Var2' := 'sBMK0'}  
{attribute 'Message.Var3' := 'sBMK1'}  
	bMeldSensFehl6	:BOOL;	

{attribute 'Message.Text' := '%Var1 hat nicht geöffnet ! (%Var2)'}		
{attribute 'Message.Info' := '}
{attribute 'Message.Type' := '7'}	
{attribute 'Message.Log'  := '1'}
{attribute 'Message.Var1' := 'sAktorName'}  
{attribute 'Message.Var2' := 'sBMK0'}  
	bLfzMeldAusg07	:BOOL;	
{attribute 'Message.Text' := '%Var1 hat nicht geschlossen ! (%Var2)'}	
{attribute 'Message.Info' := '}
{attribute 'Message.Type' := '7'}	
{attribute 'Message.Log'  := '1'}
{attribute 'Message.Var1' := 'sAktorName'}  
{attribute 'Message.Var2' := 'sBMK1'}  
	bLfzMeldAusg17	:BOOL;	
{attribute 'Message.Text' := 'Sensorfehler: %Var1 öffnen/schliessen ! (%Var2/%Var3)'}
{attribute 'Message.Info' := '}
{attribute 'Message.Type' := '8'}	
{attribute 'Message.Log'  := '1'}
{attribute 'Message.Var1' := 'sAktorName'}  
{attribute 'Message.Var2' := 'sBMK0'}  
{attribute 'Message.Var3' := 'sBMK1'}  
	bMeldSensFehl7	:BOOL;
	
{attribute 'Message.Text' := '%Var1 nicht in 0° ! (%Var2)'}		
{attribute 'Message.Info' := '}
{attribute 'Message.Type' := '7'}	
{attribute 'Message.Log'  := '1'}
{attribute 'Message.Var1' := 'sAktorName'}  
{attribute 'Message.Var2' := 'sBMK0'}  
	bLfzMeldAusg09	:BOOL;	
{attribute 'Message.Text' := '%Var1 nicht in 180° ! (%Var2)'}	
{attribute 'Message.Info' := '}
{attribute 'Message.Type' := '7'}	
{attribute 'Message.Log'  := '1'}
{attribute 'Message.Var1' := 'sAktorName'}  
{attribute 'Message.Var2' := 'sBMK1'}  
	bLfzMeldAusg19	:BOOL;	
{attribute 'Message.Text' := 'Sensorfehler: %Var1 0°/180° ! (%Var2/%Var3)'}
{attribute 'Message.Info' := '}
{attribute 'Message.Type' := '8'}	
{attribute 'Message.Log'  := '1'}
{attribute 'Message.Var1' := 'sAktorName'}  
{attribute 'Message.Var2' := 'sBMK0'}  
{attribute 'Message.Var3' := 'sBMK1'}  
	bMeldSensFehl9	:BOOL;

	sMeldText		:T_MaxString:= 'MeldText';
	sInfoText		:T_MaxString:= 'InfoText';
	sAktorName		:T_MaxString:= 'AktorName';
	sBMK0				:T_MaxString:= 'BMK0';
	sBMK1				:T_MaxString:= 'BMK1';
	sLzFehlerDef0	:T_MaxString:= 'Nicht in Def0';
	sLzFehlerDef1	:T_MaxString:= 'Nicht in Def1';
	sSensorFehlDef	:T_MaxString:= 'Def0/Def1';

END_STRUCT
END_TYPE

// DUTs/HMI_Meldungen/Meldelisten/ST_MeldAchsList
{attribute 'pack_mode' := '1'}
TYPE ST_MeldAchsList :
STRUCT

{attribute 'Message.Struct'}
	stMeldAchsfehler		:ST_MeldAchsfehler;
{attribute 'Message.Struct'}
	arrMeldAchsGruppe		:ARRAY [0..cAnzAchsGruppen] OF ST_MeldAchsGruppe;	// Fehler für Achsgruppen

END_STRUCT
END_TYPE

// DUTs/HMI_Meldungen/Meldelisten/ST_MeldEAPList
{attribute 'pack_mode' := '1'}
TYPE ST_MeldEAPList :
STRUCT

{attribute 'Message.Struct'}
	arrMeldEAPError			:ARRAY [1..cAnzEAPVerbindungen] OF ST_MeldEAPKommError;	// Meldearray für Fehler in der EAP-Kommunikationsverbindung
END_STRUCT
END_TYPE

// DUTs/HMI_Meldungen/Meldelisten/ST_MeldIOLinkList
{attribute 'pack_mode' := '1'}
TYPE ST_MeldIOLinkList :
STRUCT
	
{attribute 'Message.Struct'}
	arrMeldIOLinkKlemme	: ARRAY [0..cAnzIOLinkKlemmen] OF ST_MeldIOLinkKlemme;	// Meldearray für Fehler in den IO-Link-Klemmen
END_STRUCT
END_TYPE

// DUTs/HMI_Meldungen/Meldelisten/ST_MeldKommunikationsList
{attribute 'pack_mode' := '1'}
TYPE ST_MeldKommunikationsList :
STRUCT

{attribute 'Message.Struct'}
	arrMeldKommError			:ARRAY [1..cAnzKommError] OF ST_MeldADSKommError;	// Meldearray für Fehler in der ADS-Kommunikationsverbindung
{attribute 'Message.Struct'}
	arrMeldADS_EA_Error		:ARRAY [1..cAnzADS_EA_Error] OF ST_MeldADS_ExchangeError;	// Meldearray für Fehler in der EA-ADS-Kommunikationsverbindung
{attribute 'Message.Struct'}
	arrMeldADS_Data_Error	:ARRAY [1..cAnzADS_Data_Error] OF ST_MeldADS_ExchangeError;	// Meldearray für Fehler in der Data-ADS-Kommunikationsverbindung
END_STRUCT
END_TYPE

// DUTs/HMI_Meldungen/Meldelisten/ST_MeldPotentialList
{attribute 'pack_mode' := '1'}
TYPE ST_MeldPotentialList :
STRUCT
	
{attribute 'Message.Struct'}
	arrMeldEinspeis	:ARRAY [0..cAnzEinspeis] OF ST_MeldEinspeisKlemme;	// Meldearray für Fehler aller Einspeiseklemmen
	
{attribute 'Message.Struct'}
	arrMeldAuffrisch	:ARRAY [0..cAnzAuffrisch] OF ST_MeldAuffrischKlemme;	// Meldearray für Fehler aller Auffrischungsklemmen

END_STRUCT
END_TYPE

// DUTs/HMI_Meldungen/Meldelisten/ST_MeldSafetyList
{attribute 'pack_mode' := '1'}
TYPE ST_MeldSafetyList :
STRUCT

{attribute 'Message.Struct'}
	arrMeldGruppen			:ARRAY [0..cAnzSafetyGruppen] OF ST_MeldSafetygruppe;	// Meldearray für die Safety-Gruppen
{attribute 'Message.Struct'}
	arrMeldFBErrors		:ARRAY [0..cAnzSafetyFBError] OF ST_MeldSafetyFBErrors;	// Meldearray für die Safety-FB-Errors
{attribute 'Message.Struct'}
	arrMeldAusgang			:ARRAY [0..cAnzSafetyAusgaenge] OF ST_MeldSafetyOuts;	// Meldearray für die Safety-Ausgänge. Con-Info4 + Con-Info5
{attribute 'Message.Struct'}
	arrMeldKlemmen			:ARRAY [0..cAnzSafetyKlemmen] OF ST_MeldKlemme;	// Meldearray für die Safety-Klemmen Diagnose

END_STRUCT
END_TYPE

// DUTs/HMI_Meldungen/Meldelisten/ST_MeldSchaltSchrList
{attribute 'pack_mode' := '1'}
TYPE ST_MeldSchaltSchrList :
STRUCT
	
{attribute 'Message.Struct'}
	stMeldAusgUSV			: ST_MeldUSV;	// Meldungen für eine USV

{attribute 'Message.Struct'}
	arrMeldKlimageraet	: ARRAY [0..cAnzKlimageraete] OF ST_MeldKlimaGeraet;	// Vorgefertigte Meldungen für Klimageräte

{attribute 'Message.Struct'}
	arrMeldNetzteil		: ARRAY [0..cAnzNetzteile] OF ST_MeldSchaltNetzT;	// Vorgefertigte Meldungen für Schaltnetzteile

{attribute 'Message.Struct'}
	arrMeldSicherung		: ARRAY [0..cAnzSicherungen] OF ST_MeldSichgAutom;	// Vorgefertigte Meldungen für Sicherungsautomaten
	 
{attribute 'Message.Struct'}
	arrMeldElektSicherung	: ARRAY [0..cAnzElekSicherungen] OF ST_MeldElektrSichg;	// Vorgefertigte Meldungen für elektronische Sicherungen

{attribute 'Message.Struct'}
	arrMeldMotorschutz	: ARRAY [0..cAnzMSSchalter] OF ST_MeldMotSchutzS;	// Vorgefertigte Meldungen für Motorschutzschalter
	
{attribute 'Message.Struct'}
	arrMeldThermoueberw	: ARRAY [0..cAnzThermoueberw] OF ST_MeldThermoUeberw;	// Vorgefertigte Meldungen für thermische Überwachungen

{attribute 'Message.Struct'}
	arrBetriebsdruck		: ARRAY [0..cAnzWartungsEinheit] OF ST_MeldBetriebsdruck;	// Fehlermeldungen Betriebsdruck nicht erreicht
	
{attribute 'Message.Struct'}
	arrMeldSchaltschrHMI	: ARRAY [0..cAnzSonstige] OF ST_MeldTextAllgm;	// Vorgefertigte Meldungen. Zur freien Verfügung im Projekt.
	
END_STRUCT
END_TYPE

// DUTs/HMI_Meldungen/Meldelisten/ST_MeldSchutzberList
{attribute 'pack_mode' := '1'}
TYPE ST_MeldSchutzberList :
STRUCT

{attribute 'Message.Struct'}
	arrMeldNotHalt					:ARRAY [0..cAnzNotHalt] OF ST_MeldNotHalt;	// Meldearray für gedrückte Nothalt-Taster

{attribute 'Message.Struct'}
	arrMeldSichLichtg				:ARRAY[0..cAnzLichtgitter] OF ST_MeldSichLichtg;	// Vorgefertigte Meldungen für Lichtgitter oder Lichtschutzvorhänge

{attribute 'Message.Struct'}
	arrMeldWartgTuer				:ARRAY[0..cAnzWartungstuer] OF ST_MeldWartgTuer;	// Vorgefertigte Meldungen für Wartungstüren
	
{attribute 'Message.Struct'}
	arrMeldStHLuft					:ARRAY[0..cAnzSchutzBer] OF ST_MeldStHLuft;	// Vorgefertigte Meldungen für Wartungstüren
	
{attribute 'Message.Struct'}
	arrMeldTuerFrgBremsentest	:ARRAY[0..cAnzSchutzBer] OF ST_MeldTuerFrgBremsentest;	// Vorgefertigte Meldungen für Bremsentest
	
{attribute 'Message.Struct'}
	arrMeldSchutzbereichOffen	:ARRAY[0..cAnzSchutzBer] OF ST_MeldSchutzbereichOffen;	// Vorgefertigte Meldungen für Schutzbereich offen
	
END_STRUCT
END_TYPE

// DUTs/HMI_Meldungen/Meldelisten/ST_MeldSeriellComPort
{attribute 'pack_mode' := '1'}
TYPE ST_MeldSeriellComPort :
STRUCT

{attribute 'Message.Struct'}
	arrMeldComPortError	:ARRAY [0..cAnzComports] OF ST_MeldComPort;	// Meldearray für Fehler in den ComPorts
END_STRUCT
END_TYPE

// DUTs/HMI_Meldungen/ST_0100_Meldungen
{attribute 'pack_mode' := '1'}
TYPE ST_0100_Meldungen :
STRUCT
{attribute 'MaschPara.Name' := 'Schaltschrank'}     
{attribute 'MaschPara.TreeViewImage' 	:= '\TreeIcons\Cabinet.png'}  
	stSchaltSchr		:ST_MeldSchaltSchrList;	// Meldeliste für den Schaltschrank und alle drin befindlichen Bauteile
	
{attribute 'MaschPara.Name' := 'Schutzbereiche'}     
{attribute 'MaschPara.TreeViewImage' 	:= '\TreeIcons\Door.png'}  
	stSchutzbereiche	:ST_MeldSchutzberList;	// Meldeliste für alle Schutzbereiche, Nothalt, Lichtgitter und Schutztüren
	
{attribute 'MaschPara.Name' := 'Achsen'}   
	stAchsen				:ST_MeldAchsList;	// Meldeliste für einen allgemeinen Achsfehler und für die Achsgruppeneinspeisungen
	
{attribute 'MaschPara.Name' := 'Safety'}   
	stSafety				:ST_MeldSafetyList;	// Meldelisten für das Safetyprojekt
	
{attribute 'MaschPara.Name' := 'ADS-Kommunikation'}   
	stKommunikation	:ST_MeldKommunikationsList;	// Meldeliste für die ADS-Kommunikationsverbindung mit den anderen Anlagenteilen
	
{attribute 'MaschPara.Name' := 'EAP-Kommunikation'}   
	stEAP					:ST_MeldEAPList;	// Meldeliste für die EAP-Kommunikationsverbindung mit den anderen Anlagenteilen
	
{attribute 'MaschPara.Name' := 'Serielle-Kommunikation'}   
	stSeriellComPort	:ST_MeldSeriellComPort;	// Meldeliste für die serielle Kommunitkation über RS232
	
{attribute 'Message.Struct'}
	stDatenanf			:ST_MeldDatenanf;	// Eine Meldung für die Datenanforderung	 		 
	
{attribute 'MaschPara.Name' := 'IO-Link'}   
	stIOLink				:ST_MeldIOLinkList;	// Meldeliste für IO-Link Fehler
	
{attribute 'MaschPara.Name' := 'Einspeiseklemmen'}   
	stEinspeis			:ST_MeldPotentialList;	// Meldeliste für Potenzialeinspeisung und Auffrischung
	
{attribute 'Message.Struct'}
	stEtherCAT			:ST_MeldEtherCAT;	// Eine Meldung für die EtherCAT-Fehler
	
{attribute 'Message.Struct'}
	arrMeldEtherCAT	:ARRAY[0..cMaxAnzahlSlaveError] OF ST_MeldTextAllgm;
	
END_STRUCT
END_TYPE

// DUTs/HMI_Meldungen/ST_ParamHMIMaschine_Beispiel
// Diese Struktur soll als Beispiel und Dokumentation für die Maschinenparameter in der Avalon-HMI dienen.
// Diese Struktur kann gerne vererbt/erweitert werden oder auch nur kopiert.
// Für die Verwendung als Hauptstruktur muss eine Instanz in den Globalen Variablen angelegt werden.
// Eine andere Möglichkeit als eine Strukturinstanz wäre ein Programm- oder Funktionsbaustein.
// Die Attribute für die HMI können in 2 Varianten angegeben werden.
// Variante 1 (alte Variante) als Kommentar: stMaschParam	: ST_ParamHMIMaschine_Beispiel;	// @1: Name @2: Einheit @3: Min-Wert @4: Max-Wert @8: Var-Update als BOOL @9: Infotext @10: UserLever (Obsolet) @11: +-1, +-2, usw. Verschieben des TreeViewItem @12: Name des TreeViewItem aus 11 13@: Pfad zum Icon
// Variante 2 mit Attributen :
//{attribute 'MaschPara.Name'} Name
//{attribute 'MaschPara.Type'} Einheit
//{attribute 'MaschPara.Min'} Min-Wert
//{attribute 'MaschPara.Max'} Max-Wert
//{attribute 'MaschPara.ReactOnPlcPropertyChanged'} Var-Update als BOOL
//{attribute 'MaschPara.Info'} Infotext
//{attribute 'MaschPara.TreeViewLayer'} +-1, +-2, usw. Verschieben des TreeViewItem
//{attribute 'MaschPara.TreeViewDesc'} Name des TreeViewItem aus 11
//{attribute 'MaschPara.TreeViewImage'} Pfad zum Icon
//{attribute 'MaschPara.LanguageKeyText'} Sprechumschaltung. sLanguageKeyText muss in Struktur definiert sein
//{attribute 'DesignerControl.ControlType'} Hiermit können definierte oder Standard Controls in der HMI geladen werden
// Standard-Controls:
// System.Windows.Controls.Label
// System.Windows.Controls.TextBox
// System.Windows.Controls.Button
// System.Windows.Controls.CheckBox
// System.Windows.Controls.Image
// System.Windows.Controls.Border
// System.Windows.Controls.ComboBox
// System.Windows.Controls.ListBox
// System.Windows.Controls.RadioButton
// System.Windows.Controls.TextBlock
// System.Windows.Controls.ToggleButton
// Beckhoff.App.Base.WPF.Controls.DataGrid.BADataGrid
// Beckhoff.App.Product.PlcHmiDesigner.Controls.ErrorFlag.ErrorFlag
// Beckhoff.App.Product.PlcHmiDesigner.Controls.NavigationControl.NavigationControl
{attribute 'pack_mode' := '1'}
TYPE ST_ParamHMIMaschine_Beispiel :
STRUCT
	//arrParam_Achsen				:ARRAY[1..cAnzAchsenReal] OF ST_ParamAchsen;			(*@1: Servo-Achsen *)
	//stParam_FUs					:ST_ParamFrequenzumrichter;								(*@1: Frequenzumrichter	*)
	
	// Beispiele für Parameter nach Variante 1
	//stParam_DrehshutlleEinl	:ST_ParamDrehshutlleEinl;									(*@1: P4100 Drehshuttle Einlauf					*)	
	//stParam_SpannStation		:ST_ParamSpannSt;												(*@1: P4200 Spannstation							*)
	//stParam_Hauptpresse		:ST_ParamPresse;												(*@1: P4400 Hauptpresse								*)
	//stParam_RueckwSchr			:ST_ParamRwSchrauber;										(*@1: P4460 Rückwand-Schrauber 					*)
	//stParam_WAufhSchr			:ST_ParamWASchrauber;										(*@1: P4440/P4450 Wandaufhänger-Schrauber 	*)
	//stParam_DrehshutlleAusl	:ST_ParamDrehshutlleAusl;									(*@1: P4600 Drehshuttle Auslauf					*)
	//nAnlagenNummer				:INT;	// @1: Anlagenteil @3: 1 @4: 5 @9: Das ist die Nummer des Anlagenteils
	
	// Beispiele für Parameter nach Variant 2
	//{attribute 'MaschPara.Name' := 'Maschinename'}
	//{attribute 'MaschPara.Info' := 'Das ist der Name der Maschine'}
	//{attribute 'MaschPara.LanguageKeyText' := 'True'}
	//{attribute 'MaschPara.TreeViewImage' := '\TreeIcons\Kacheln.png'}
	//sNameDerMaschine			:STRING;
	
	//{attribute 'MaschPara.Name' := 'Anlagenteil'}
	//{attribute 'MaschPara.Min'	:= '1'}
	//{attribute 'MaschPara.Max' := '5'}
	//{attribute 'MaschPara.Info' := 'Das ist die Nummer des Anlagenteils'}
	//{attribute 'MaschPara.LanguageKeyText' := 'True'}
	//{attribute 'MaschPara.TreeViewImage' := '\TreeIcons\Kacheln.png'}
	//nAnlagenNummer				:INT;

	// Diese Variablen müssen in den Einstellungen der HMI angegeben werden
	bStartWriteFromHMI		:BOOL;	// PLC->HMI HMI soll die Maschinendaten schreiben
	bQuittWriteFromHMI		:BOOL;	// HMI->PLC HMI hat die Maschinendaten fertig geschrieben
	bStartReadFromHMI			:BOOL;	// PLC_>HMI HMI soll Maschinendaten neu einlesen
	sActFilenameHMI			:STRING;	// Aktueller Dateiname von der Maschinenparameter-Datei
END_STRUCT
END_TYPE

// DUTs/HMI_Parameter/ST_UniAchsAnstgParam
// Diese Struktur deklariert Parameter für den UniAchsAnstg-Baustein.
// Verwendung der Presets: {attribute 'Preset.GeschwMin' := '@.fMinGeschwindigkeit'}
// oder dirket als Zahl: {attribute 'Preset.GeschwMin' := '10'}
// muss über der Instanz von ST_UniAchsAnstgParam stehen
// mögliche Presets: 'Preset.GeschwMin', 'Preset.GeschwMax'
// dazu kommt noch ein Preset für die Gruppierung der Parameter, also eine Überschrift.
// dieses wird so verwender: {attribute 'Preset.GroupName' := 'Hier ein Gruppenname'}
// der Gruppenname kann auch mit @.XXX eine globale Variable oder eine Variable in der folgenden Instantz der Struktur sein.
{attribute 'pack_mode' := '1'}
TYPE ST_UniAchsAnstgParam :
STRUCT
// Verwendung der Presets: {attribute 'Preset.GeschwMin' := '@.fMinGeschwindigkeit'}
// oder dirket als Zahl: {attribute 'Preset.GeschwMin' := '10'}
// muss über der Instanz von ST_UniAchsAnstgParam stehen
// mögliche Presets: 'Preset.GeschwMin', 'Preset.GeschwMax'
//{attribute 'MaschPara.Margin' := '0 20 0 0'}	
{attribute 'MaschPara.Name' := 'Geschwindigkeitsvorgabe'}
{attribute 'MaschPara.Type' := '%'}
{attribute 'MaschPara.Min' := 'Preset.GeschwMin'}
{attribute 'MaschPara.Max' := 'Preset.GeschwMax'}
{attribute 'MaschPara.Info' := 'Geschwindigkeitsvorgabe'}
{attribute 'MaschPara.TreeViewLayer' := '-1'}
{attribute 'MaschPara.GroupName' := 'Preset.GroupName'}
	fGeschwVorg		:LREAL;

// Verwendung der Presets: {attribute 'Preset.PosGrdstlgMin' := '@.fMinGrundstellung'}
// oder dirket als Zahl: {attribute 'Preset.PosGrdstlgMin' := '10'}
// muss über der Instanz von ST_UniAchsAnstgParam stehen
// mögliche Presets: 'Preset.PosGrdstlgMin', 'Preset.PosGrdstlgMax'
{attribute 'MaschPara.Name' := 'Grundposition'}
{attribute 'MaschPara.Type' := 'mm'}
{attribute 'MaschPara.Min' := 'Preset.PosGrdstlgMin'}
{attribute 'MaschPara.Max' := 'Preset.PosGrdstlgMax'}
{attribute 'MaschPara.Info' := 'Grundposition'}
{attribute 'MaschPara.TreeViewLayer' := '-1'}
{attribute 'MaschPara.GroupName' := 'Preset.GroupName'}
	fGrdstlgPos		:LREAL;

// Verwendung der Presets: {attribute 'Preset.PosParkMin' := '@.fMinParkpos'}
// oder dirket als Zahl: {attribute 'Preset.PosParkMin' := '10'}
// muss über der Instanz von ST_UniAchsAnstgParam stehen
// mögliche Presets: 'Preset.PosParkMin', 'Preset.PosParkMax'	
{attribute 'MaschPara.Name' := 'Parkposition'}
{attribute 'MaschPara.Type' := 'mm'}
{attribute 'MaschPara.Min' := 'Preset.PosParkMin'}
{attribute 'MaschPara.Max' := 'Preset.PosParkMax'}
{attribute 'MaschPara.Info' := 'Parkposition'}
{attribute 'MaschPara.TreeViewLayer' := '-1'}
{attribute 'MaschPara.GroupName' := 'Preset.GroupName'}
	fParkPos			:LREAL;

// Verwendung der Presets: {attribute 'Preset.PosReferenzMin' := '@.fMinRefpos'}
// oder dirket als Zahl: {attribute 'Preset.PosReferenzMin' := '10'}
// muss über der Instanz von ST_UniAchsAnstgParam stehen
// mögliche Presets: 'Preset.PosReferenzMin', 'Preset.PosReferenzMax'		
{attribute 'MaschPara.Name' := 'Referenzposition Encoder'}
{attribute 'MaschPara.Type' := 'mm'}
{attribute 'MaschPara.Min' := 'Preset.PosReferenzMin'}
{attribute 'MaschPara.Max' := 'Preset.PosReferenzMax'}
{attribute 'MaschPara.Info' := 'Referenzposition Encoder'}
{attribute 'MaschPara.TreeViewLayer' := '-1'}
{attribute 'MaschPara.GroupName' := 'Preset.GroupName'}
	fReferenzPos	:LREAL;

END_STRUCT
END_TYPE

// DUTs/HMI_Parameter/ST_UniAntrAnstgParamAggr
// Diese Struktur deklariert Parameter für den UniAnstgSEW-Baustein wenn dieser als Aggregat (z.B. Bohraggregat) genutzt wird.
// Zusätzlich zu den Aggregat-Parameter kommen hier noch die Hochlaufparamter hinzu.
// Verwendung der Presets: {attribute 'Preset.GeschwMin' := '@.fMinGeschwindigkeitVMin'}
// oder dirket als Zahl: {attribute 'Preset.GeschwMin' := '10'}
// muss über der Instanz von ST_UniAntrAnstgParamAggr stehen
// mögliche Presets: 'Preset.GeschwMin', 'Preset.GeschwMax'
// dazu kommt noch ein Preset für die Gruppierung der Parameter, also eine Überschrift.
// dieses wird so verwender: {attribute 'Preset.GroupName' := 'Hier ein Gruppenname'}
// der Gruppenname kann auch mit @.XXX eine globale Variable oder eine Variable in der folgenden Instantz der Struktur sein.
{attribute 'pack_mode' := '1'}
TYPE ST_UniAntrAnstgParamAggr :
STRUCT
// Verwendung der Presets: {attribute 'Preset.GeschwMin' := '@.fMinGeschwindigkeitVMin'}
// oder dirket als Zahl: {attribute 'Preset.GeschwMin' := '10'}
// muss über der Instanz von ST_UniAntrAnstgParamAggr stehen
// mögliche Presets: 'Preset.GeschwMin', 'Preset.GeschwMax'
//{attribute 'MaschPara.Margin' := '0 20 0 0'}	
{attribute 'MaschPara.Name' := 'minimale Geschwindigkeit'}
{attribute 'MaschPara.Type' := '%'}
{attribute 'MaschPara.Min' := 'Preset.GeschwMin'}
{attribute 'MaschPara.Max' := 'Preset.GeschwMax'}
{attribute 'MaschPara.Info' := 'minimale Geschwindigkeit'}		
{attribute 'MaschPara.TreeViewLayer' := '-1'}
{attribute 'MaschPara.GroupName' := 'Preset.GroupName'}
	fVmin		:LREAL;
// Verwendung der Presets: {attribute 'Preset.GeschwMin' := '@.fMinGeschwindigkeitVMax'}
// oder dirket als Zahl: {attribute 'Preset.GeschwMin' := '10'}
// muss über der Instanz von ST_UniAntrAnstgParamAggr stehen
// mögliche Presets: 'Preset.GeschwMin', 'Preset.GeschwMax'
{attribute 'MaschPara.Name' := 'maximale Geschwindigkeit'}
{attribute 'MaschPara.Type' := '%'}
{attribute 'MaschPara.Min' := 'Preset.GeschwMin'}
{attribute 'MaschPara.Max' := 'Preset.GeschwMax'}
{attribute 'MaschPara.Info' := 'maximale Geschwindigkeit'}	
{attribute 'MaschPara.TreeViewLayer' := '-1'}
{attribute 'MaschPara.GroupName' := 'Preset.GroupName'}
	fVmax		:LREAL;
// Verwendung der Presets: {attribute 'Preset.GeschwMin' := '@.fMinGeschwindigkeitV1'}
// oder dirket als Zahl: {attribute 'Preset.GeschwMin' := '10'}
// muss über der Instanz von ST_UniAntrAnstgParamAggr stehen
// mögliche Presets: 'Preset.GeschwMin', 'Preset.GeschwMax'
{attribute 'MaschPara.Name' := 'Geschwindigkeit 1'}
{attribute 'MaschPara.Type' := '%'}
{attribute 'MaschPara.Min' := 'Preset.GeschwMin'}
{attribute 'MaschPara.Max' := 'Preset.GeschwMax'}
{attribute 'MaschPara.Info' := 'Geschwindigkeit 1'}
{attribute 'MaschPara.TreeViewLayer' := '-1'}
{attribute 'MaschPara.GroupName' := 'Preset.GroupName'}
	fV_1		:LREAL;	
// Verwendung der Presets: {attribute 'Preset.GeschwMin' := '@.fMinGeschwindigkeitV2'}
// oder dirket als Zahl: {attribute 'Preset.GeschwMin' := '10'}
// muss über der Instanz von ST_UniAntrAnstgParamAggr stehen
// mögliche Presets: 'Preset.GeschwMin', 'Preset.GeschwMax'
{attribute 'MaschPara.Name' := 'Geschwindigkeit 2'}
{attribute 'MaschPara.Type' := '%'}
{attribute 'MaschPara.Min' := 'Preset.GeschwMin'}
{attribute 'MaschPara.Max' := 'Preset.GeschwMax'}
{attribute 'MaschPara.Info' := 'Geschwindigkeit 2'}	
{attribute 'MaschPara.TreeViewLayer' := '-1'}
{attribute 'MaschPara.GroupName' := 'Preset.GroupName'}
	fV_2		:LREAL;	
// Verwendung der Presets: {attribute 'Preset.GeschwMin' := '@.fMinGeschwindigkeitV3'}
// oder dirket als Zahl: {attribute 'Preset.GeschwMin' := '10'}
// muss über der Instanz von ST_UniAntrAnstgParamAggr stehen
// mögliche Presets: 'Preset.GeschwMin', 'Preset.GeschwMax'
{attribute 'MaschPara.Name' := 'Geschwindigkeit 3'}
{attribute 'MaschPara.Type' := '%'}
{attribute 'MaschPara.Min' := 'Preset.GeschwMin'}
{attribute 'MaschPara.Max' := 'Preset.GeschwMax'}
{attribute 'MaschPara.Info' := 'Geschwindigkeit 3'}	
{attribute 'MaschPara.TreeViewLayer' := '-1'}
{attribute 'MaschPara.GroupName' := 'Preset.GroupName'}
	fV_3		:LREAL;
// Verwendung der Presets: {attribute 'Preset.RampeMin' := '@.fMinRampeAb'}
// oder dirket als Zahl: {attribute 'Preset.RampeMin' := '10'}
// muss über der Instanz von ST_UniAntrAnstgParamAggr stehen
// mögliche Presets: 'Preset.RampeMin', 'Preset.RampeMax'
{attribute 'MaschPara.Name' := 'Verzögerungs-Rampe'}
{attribute 'MaschPara.Type' := 'ms'}
{attribute 'MaschPara.Min' := 'Preset.RampeMin'}
{attribute 'MaschPara.Max' := 'Preset.RampeMax'}
{attribute 'MaschPara.Info' := 'Verzögerungs-Rampe'}	
{attribute 'MaschPara.TreeViewLayer' := '-1'}
{attribute 'MaschPara.GroupName' := 'Preset.GroupName'}
	fRampe_ab:LREAL;
// Verwendung der Presets: {attribute 'Preset.RampeMin' := '@.fMinRampeAuf'}
// oder dirket als Zahl: {attribute 'Preset.RampeMin' := '10'}
// muss über der Instanz von ST_UniAntrAnstgParamAggr stehen
// mögliche Presets: 'Preset.RampeMin', 'Preset.RampeMax'
{attribute 'MaschPara.Name' := 'Beschleunigungs-Rampe'}
{attribute 'MaschPara.Type' := 'ms'}
{attribute 'MaschPara.Min' := 'Preset.RampeMin'}
{attribute 'MaschPara.Max' := 'Preset.RampeMax'}
{attribute 'MaschPara.Info' := 'Beschleunigungs-Rampe'}	
{attribute 'MaschPara.TreeViewLayer' := '-1'}
{attribute 'MaschPara.GroupName' := 'Preset.GroupName'}
	fRampe_auf:LREAL;
	
END_STRUCT
END_TYPE

// DUTs/HMI_Parameter/ST_UniAntrAnstgParamAggrHF
// Diese Struktur deklariert Parameter für den UniAnstgSEW-Baustein wenn dieser als Aggregat genutzt wird.
// Verwendung der Presets: {attribute 'Preset.GeschwMin' := '@.fMinGeschwindigkeitVMin'}
// oder dirket als Zahl: {attribute 'Preset.GeschwMin' := '10'}
// muss über der Instanz von ST_UniAntrAnstgParamAggrHF stehen
// mögliche Presets: 'Preset.GeschwMin', 'Preset.GeschwMax'
// dazu kommt noch ein Preset für die Gruppierung der Parameter, also eine Überschrift.
// dieses wird so verwender: {attribute 'Preset.GroupName' := 'Hier ein Gruppenname'}
// der Gruppenname kann auch mit @.XXX eine globale Variable oder eine Variable in der folgenden Instantz der Struktur sein.
{attribute 'pack_mode' := '1'}
TYPE ST_UniAntrAnstgParamAggrHF :
STRUCT
// Verwendung der Presets: {attribute 'Preset.GeschwMin' := '@.fMinGeschwindigkeitVMin'}
// oder dirket als Zahl: {attribute 'Preset.GeschwMin' := '10'}
// muss über der Instanz von ST_UniAntrAnstgParamAggrHF stehen
// mögliche Presets: 'Preset.GeschwMin', 'Preset.GeschwMax'
//{attribute 'MaschPara.Margin' := '0 20 0 0'}	
{attribute 'MaschPara.Name' := 'minimale Geschwindigkeit'}
{attribute 'MaschPara.Type' := '%'}
{attribute 'MaschPara.Min' := 'Preset.GeschwMin'}
{attribute 'MaschPara.Max' := 'Preset.GeschwMax'}
{attribute 'MaschPara.Info' := 'minimale Geschwindigkeit'}		
{attribute 'MaschPara.TreeViewLayer' := '-1'}
{attribute 'MaschPara.GroupName' := 'Preset.GroupName'}
	fVmin		:LREAL;
// Verwendung der Presets: {attribute 'Preset.GeschwMin' := '@.fMinGeschwindigkeitVMax'}
// oder dirket als Zahl: {attribute 'Preset.GeschwMin' := '10'}
// muss über der Instanz von ST_UniAntrAnstgParamAggrHF stehen
// mögliche Presets: 'Preset.GeschwMin', 'Preset.GeschwMax'
{attribute 'MaschPara.Name' := 'maximale Geschwindigkeit'}
{attribute 'MaschPara.Type' := '%'}
{attribute 'MaschPara.Min' := 'Preset.GeschwMin'}
{attribute 'MaschPara.Max' := 'Preset.GeschwMax'}
{attribute 'MaschPara.Info' := 'maximale Geschwindigkeit'}	
{attribute 'MaschPara.TreeViewLayer' := '-1'}
{attribute 'MaschPara.GroupName' := 'Preset.GroupName'}
	fVmax		:LREAL;
// Verwendung der Presets: {attribute 'Preset.GeschwMin' := '@.fMinGeschwindigkeitV1'}
// oder dirket als Zahl: {attribute 'Preset.GeschwMin' := '10'}
// muss über der Instanz von ST_UniAntrAnstgParamAggrHF stehen
// mögliche Presets: 'Preset.GeschwMin', 'Preset.GeschwMax'
{attribute 'MaschPara.Name' := 'Geschwindigkeit 1'}
{attribute 'MaschPara.Type' := '%'}
{attribute 'MaschPara.Min' := 'Preset.GeschwMin'}
{attribute 'MaschPara.Max' := 'Preset.GeschwMax'}
{attribute 'MaschPara.Info' := 'Geschwindigkeit 1'}
{attribute 'MaschPara.TreeViewLayer' := '-1'}
{attribute 'MaschPara.GroupName' := 'Preset.GroupName'}
	fV_1		:LREAL;	
// Verwendung der Presets: {attribute 'Preset.GeschwMin' := '@.fMinGeschwindigkeitV2'}
// oder dirket als Zahl: {attribute 'Preset.GeschwMin' := '10'}
// muss über der Instanz von ST_UniAntrAnstgParamAggrHF stehen
// mögliche Presets: 'Preset.GeschwMin', 'Preset.GeschwMax'
{attribute 'MaschPara.Name' := 'Geschwindigkeit 2'}
{attribute 'MaschPara.Type' := '%'}
{attribute 'MaschPara.Min' := 'Preset.GeschwMin'}
{attribute 'MaschPara.Max' := 'Preset.GeschwMax'}
{attribute 'MaschPara.Info' := 'Geschwindigkeit 2'}	
{attribute 'MaschPara.TreeViewLayer' := '-1'}
{attribute 'MaschPara.GroupName' := 'Preset.GroupName'}
	fV_2		:LREAL;	
// Verwendung der Presets: {attribute 'Preset.GeschwMin' := '@.fMinGeschwindigkeitV3'}
// oder dirket als Zahl: {attribute 'Preset.GeschwMin' := '10'}
// muss über der Instanz von ST_UniAntrAnstgParamAggrHF stehen
// mögliche Presets: 'Preset.GeschwMin', 'Preset.GeschwMax'
{attribute 'MaschPara.Name' := 'Geschwindigkeit 3'}
{attribute 'MaschPara.Type' := '%'}
{attribute 'MaschPara.Min' := 'Preset.GeschwMin'}
{attribute 'MaschPara.Max' := 'Preset.GeschwMax'}
{attribute 'MaschPara.Info' := 'Geschwindigkeit 3'}	
{attribute 'MaschPara.TreeViewLayer' := '-1'}
{attribute 'MaschPara.GroupName' := 'Preset.GroupName'}
	fV_3		:LREAL;
// Verwendung der Presets: {attribute 'Preset.RampeMin' := '@.fMinRampeAb'}
// oder dirket als Zahl: {attribute 'Preset.RampeMin' := '10'}
// muss über der Instanz von ST_UniAntrAnstgParamAggrHF stehen
// mögliche Presets: 'Preset.RampeMin', 'Preset.RampeMax'
{attribute 'MaschPara.Name' := 'Verzögerungs-Rampe'}
{attribute 'MaschPara.Type' := 'ms'}
{attribute 'MaschPara.Min' := 'Preset.RampeMin'}
{attribute 'MaschPara.Max' := 'Preset.RampeMax'}
{attribute 'MaschPara.Info' := 'Verzögerungs-Rampe'}	
{attribute 'MaschPara.TreeViewLayer' := '-1'}
{attribute 'MaschPara.GroupName' := 'Preset.GroupName'}
	fRampe_ab:LREAL;
// Verwendung der Presets: {attribute 'Preset.RampeMin' := '@.fMinRampeAuf'}
// oder dirket als Zahl: {attribute 'Preset.RampeMin' := '10'}
// muss über der Instanz von ST_UniAntrAnstgParamAggrHF stehen
// mögliche Presets: 'Preset.RampeMin', 'Preset.RampeMax'
{attribute 'MaschPara.Name' := 'Beschleunigungs-Rampe'}
{attribute 'MaschPara.Type' := 'ms'}
{attribute 'MaschPara.Min' := 'Preset.RampeMin'}
{attribute 'MaschPara.Max' := 'Preset.RampeMax'}
{attribute 'MaschPara.Info' := 'Beschleunigungs-Rampe'}	
{attribute 'MaschPara.TreeViewLayer' := '-1'}
{attribute 'MaschPara.GroupName' := 'Preset.GroupName'}
	fRampe_auf:LREAL;

